C07265=1069.427,-106.395,-57.676,172.308,22.663,154.150
C07266=1069.421,-106.645,-57.666,172.306,22.662,154.150
C07267=1069.415,-106.895,-57.656,172.305,22.661,154.150
C07268=1069.408,-107.144,-57.646,172.303,22.660,154.150
C07269=1069.402,-107.394,-57.636,172.302,22.659,154.150
C07270=1069.396,-107.644,-57.627,172.300,22.658,154.150
C07271=1069.390,-107.894,-57.617,172.299,22.657,154.150
C07272=1069.385,-108.144,-57.607,172.297,22.655,154.150
C07273=1069.378,-108.393,-57.597,172.295,22.654,154.150
C07274=1069.372,-108.643,-57.587,172.294,22.653,154.151
C07275=1069.366,-108.893,-57.578,172.292,22.652,154.151
C07276=1069.360,-109.142,-57.568,172.290,22.651,154.150
C07277=1069.353,-109.392,-57.559,172.289,22.650,154.151
C07278=1069.347,-109.642,-57.549,172.287,22.648,154.151
C07279=1069.341,-109.891,-57.539,172.285,22.648,154.151
C07280=1069.335,-110.141,-57.529,172.284,22.646,154.151
C07281=1069.329,-110.391,-57.519,172.282,22.646,154.151
C07282=1069.323,-110.641,-57.509,172.280,22.644,154.151
C07283=1069.317,-110.891,-57.500,172.279,22.643,154.151
C07284=1069.311,-111.141,-57.490,172.277,22.642,154.151
C07285=1069.304,-111.390,-57.481,172.275,22.641,154.151
C07286=1069.298,-111.640,-57.470,172.273,22.640,154.151
C07287=1069.292,-111.889,-57.461,172.272,22.639,154.151
C07288=1069.286,-112.139,-57.451,172.270,22.638,154.151
C07289=1069.279,-112.389,-57.442,172.268,22.636,154.151
C07290=1069.273,-112.639,-57.432,172.267,22.636,154.151
C07291=1069.267,-112.889,-57.423,172.265,22.634,154.151
C07292=1069.261,-113.138,-57.413,172.263,22.634,154.151
C07293=1069.255,-113.388,-57.403,172.261,22.632,154.151
C07294=1069.250,-113.638,-57.394,172.260,22.631,154.151
C07295=1069.242,-113.918,-57.383,172.258,22.630,154.151
C07296=1069.236,-114.198,-57.373,172.256,22.629,154.151
C07297=1069.229,-114.478,-57.361,172.255,22.628,154.151
C07298=1069.222,-114.758,-57.351,172.253,22.627,154.151
C07299=1069.216,-115.008,-57.341,172.251,22.626,154.152
C07300=1069.210,-115.258,-57.332,172.249,22.625,154.152
C07301=1069.204,-115.508,-57.322,172.248,22.624,154.152
C07302=1069.198,-115.757,-57.312,172.246,22.623,154.152
C07303=1069.191,-116.007,-57.303,172.244,22.622,154.152
C07304=1069.185,-116.257,-57.293,172.243,22.621,154.152
C07305=1069.179,-116.507,-57.284,172.241,22.620,154.152
C07306=1069.173,-116.757,-57.274,172.239,22.619,154.152
C07307=1069.166,-117.006,-57.265,172.237,22.618,154.152
C07308=1069.160,-117.256,-57.256,172.236,22.617,154.152
C07309=1069.154,-117.505,-57.246,172.234,22.616,154.152
C07310=1069.148,-117.755,-57.237,172.232,22.615,154.152
C07311=1069.142,-118.005,-57.227,172.231,22.614,154.152
C07312=1069.136,-118.254,-57.218,172.229,22.613,154.152
C07313=1069.130,-118.504,-57.208,172.227,22.612,154.153
C07314=1069.123,-118.754,-57.199,172.226,22.611,154.152
C07315=1069.117,-119.004,-57.189,172.225,22.610,154.153
C07316=1069.111,-119.254,-57.179,172.223,22.610,154.153
C07317=1069.105,-119.504,-57.171,172.221,22.608,154.153
C07318=1069.100,-119.753,-57.161,172.219,22.607,154.153
C07319=1069.093,-120.003,-57.152,172.218,22.607,154.153
C07320=1069.087,-120.252,-57.143,172.216,22.606,154.153
C07321=1069.080,-120.502,-57.133,172.214,22.605,154.153
C07322=1069.074,-120.752,-57.124,172.212,22.604,154.153
C07323=1069.068,-121.002,-57.114,172.211,22.603,154.153
C07324=1069.062,-121.252,-57.105,172.209,22.602,154.153
C07325=1069.057,-121.501,-57.096,172.207,22.601,154.153
C07326=1069.050,-121.751,-57.087,172.205,22.600,154.153
C07327=1069.043,-122.001,-57.078,172.204,22.599,154.154
C07328=1069.037,-122.250,-57.068,172.202,22.599,154.154
C07329=1069.031,-122.500,-57.058,172.200,22.597,154.154
C07330=1069.025,-122.751,-57.050,172.199,22.597,154.154
C07331=1069.019,-123.000,-57.040,172.197,22.596,154.154
C07332=1069.014,-123.250,-57.031,172.196,22.595,154.154
C07333=1069.007,-123.499,-57.022,172.194,22.594,154.154
C07334=1069.000,-123.749,-57.012,172.192,22.593,154.154
C07335=1068.995,-123.999,-57.003,172.190,22.592,154.154
C07336=1068.988,-124.249,-56.994,172.189,22.592,154.154
C07337=1068.983,-124.498,-56.985,172.187,22.591,154.154
C07338=1068.976,-124.748,-56.976,172.185,22.590,154.155
C07339=1068.970,-124.998,-56.967,172.183,22.589,154.155
C07340=1068.964,-125.248,-56.957,172.182,22.588,154.155
C07341=1068.958,-125.498,-56.948,172.180,22.587,154.155
C07342=1068.951,-125.747,-56.939,172.178,22.586,154.155
C07343=1068.946,-125.997,-56.930,172.177,22.586,154.155
C07344=1068.939,-126.247,-56.921,172.175,22.585,154.155
C07345=1068.933,-126.496,-56.911,172.174,22.584,154.155
C07346=1068.927,-126.747,-56.903,172.172,22.584,154.155
C07347=1068.920,-126.996,-56.893,172.170,22.583,154.155
C07348=1068.915,-127.245,-56.884,172.168,22.582,154.156
C07349=1068.908,-127.495,-56.875,172.166,22.581,154.156
C07350=1068.902,-127.745,-56.866,172.165,22.580,154.156
C07351=1068.897,-127.996,-56.857,172.163,22.580,154.156
C07352=1068.893,-128.247,-56.847,172.161,22.578,154.156
C07353=1068.890,-128.498,-56.836,172.160,22.575,154.155
C07354=1068.890,-128.748,-56.824,172.159,22.573,154.155
C07355=1068.892,-129.001,-56.811,172.158,22.569,154.155
C07356=1068.896,-129.253,-56.798,172.158,22.565,154.154
C07357=1068.901,-129.505,-56.784,172.158,22.560,154.153
C07358=1068.908,-129.755,-56.769,172.158,22.554,154.152
C07359=1068.520,-129.777,-56.938,172.111,22.697,154.184
C07360=1068.512,-129.527,-56.954,172.111,22.703,154.185
C07361=1068.506,-129.276,-56.969,172.111,22.708,154.186
C07362=1068.503,-129.023,-56.982,172.112,22.712,154.187
C07363=1068.501,-128.771,-56.995,172.113,22.716,154.188
C07364=1068.501,-128.520,-57.006,172.114,22.719,154.188
C07365=1068.503,-128.270,-57.017,172.114,22.722,154.188
C07366=1068.507,-128.019,-57.027,172.116,22.723,154.188
C07367=1068.513,-127.768,-57.036,172.117,22.724,154.188
C07368=1068.519,-127.518,-57.046,172.119,22.725,154.188
C07369=1068.525,-127.268,-57.054,172.121,22.726,154.188
C07370=1068.532,-127.018,-57.064,172.123,22.727,154.188
C07371=1068.538,-126.768,-57.073,172.125,22.727,154.188
C07372=1068.543,-126.519,-57.083,172.126,22.728,154.188
C07373=1068.550,-126.269,-57.091,172.128,22.729,154.188
C07374=1068.556,-126.019,-57.100,172.130,22.730,154.188
C07375=1068.562,-125.770,-57.110,172.132,22.730,154.188
C07376=1068.569,-125.519,-57.118,172.133,22.731,154.187
C07377=1068.574,-125.270,-57.127,172.135,22.732,154.187
C07378=1068.581,-125.021,-57.137,172.136,22.732,154.187
C07379=1068.587,-124.771,-57.147,172.138,22.733,154.187
C07380=1068.593,-124.521,-57.155,172.140,22.734,154.187
C07381=1068.600,-124.271,-57.164,172.141,22.735,154.187
C07382=1068.606,-124.021,-57.174,172.143,22.736,154.187
C07383=1068.611,-123.772,-57.183,172.145,22.737,154.187
C07384=1068.617,-123.522,-57.192,172.147,22.738,154.187
C07385=1068.623,-123.272,-57.202,172.149,22.738,154.187
C07386=1068.630,-123.022,-57.211,172.150,22.740,154.187
C07387=1068.636,-122.772,-57.220,172.152,22.740,154.186
C07388=1068.642,-122.523,-57.229,172.154,22.741,154.186
C07389=1068.648,-122.273,-57.238,172.156,22.742,154.186
C07390=1068.654,-122.023,-57.248,172.157,22.743,154.186
C07391=1068.660,-121.773,-57.257,172.159,22.744,154.186
C07392=1068.667,-121.524,-57.266,172.161,22.745,154.186
C07393=1068.673,-121.274,-57.276,172.163,22.746,154.186
C07394=1068.679,-121.024,-57.285,172.164,22.746,154.186
C07395=1068.685,-120.775,-57.294,172.165,22.747,154.186
C07396=1068.691,-120.525,-57.303,172.167,22.748,154.186
C07397=1068.697,-120.275,-57.313,172.169,22.749,154.186
C07398=1068.703,-120.025,-57.323,172.171,22.750,154.186
C07399=1068.709,-119.775,-57.332,172.172,22.751,154.186
C07400=1068.716,-119.526,-57.341,172.174,22.752,154.185
C07401=1068.722,-119.276,-57.351,172.176,22.753,154.185
C07402=1068.728,-119.027,-57.360,172.177,22.754,154.185
C07403=1068.734,-118.777,-57.369,172.179,22.755,154.185
C07404=1068.740,-118.527,-57.378,172.181,22.755,154.185
C07405=1068.746,-118.277,-57.388,172.183,22.757,154.185
C07406=1068.752,-118.027,-57.397,172.184,22.758,154.185
C07407=1068.759,-117.777,-57.407,172.186,22.758,154.185
C07408=1068.765,-117.528,-57.417,172.188,22.760,154.185
C07409=1068.771,-117.278,-57.426,172.190,22.760,154.185
C07410=1068.777,-117.028,-57.436,172.191,22.761,154.185
C07411=1068.783,-116.778,-57.445,172.193,22.763,154.185
C07412=1068.789,-116.528,-57.455,172.194,22.763,154.185
C07413=1068.795,-116.279,-57.464,172.195,22.764,154.185
C07414=1068.801,-116.029,-57.474,172.197,22.765,154.184
C07415=1068.808,-115.780,-57.483,172.199,22.766,154.184
C07416=1068.814,-115.530,-57.492,172.201,22.767,154.184
C07417=1068.820,-115.280,-57.502,172.203,22.768,154.184
C07418=1068.827,-115.031,-57.511,172.204,22.769,154.184
C07419=1068.833,-114.781,-57.521,172.206,22.770,154.184
C07420=1068.840,-114.500,-57.532,172.208,22.771,154.184
C07421=1068.846,-114.220,-57.543,172.210,22.773,154.184
C07422=1068.853,-113.940,-57.554,172.212,22.774,154.184
C07423=1068.860,-113.660,-57.564,172.214,22.775,154.184
C07424=1068.866,-113.410,-57.574,172.215,22.776,154.184
C07425=1068.872,-113.160,-57.584,172.217,22.777,154.184
C07426=1068.878,-112.910,-57.593,172.219,22.778,154.184
C07427=1068.884,-112.661,-57.603,172.220,22.779,154.184
C07428=1068.891,-112.411,-57.612,172.222,22.780,154.184
C07429=1068.897,-112.161,-57.622,172.224,22.781,154.184
C07430=1068.903,-111.911,-57.631,172.226,22.782,154.184
C07431=1068.909,-111.661,-57.641,172.227,22.783,154.184
C07432=1068.916,-111.412,-57.651,172.229,22.784,154.184
C07433=1068.922,-111.162,-57.661,172.231,22.786,154.184
C07434=1068.927,-110.912,-57.671,172.232,22.787,154.183
C07435=1068.933,-110.662,-57.681,172.234,22.788,154.183
C07436=1068.939,-110.413,-57.690,172.235,22.788,154.183
C07437=1068.946,-110.163,-57.700,172.236,22.790,154.183
C07438=1068.952,-109.913,-57.709,172.238,22.790,154.183
C07439=1068.958,-109.664,-57.720,172.240,22.792,154.183
C07440=1068.964,-109.414,-57.729,172.242,22.793,154.183
C07441=1068.971,-109.164,-57.739,172.243,22.794,154.183
C07442=1068.977,-108.915,-57.748,172.245,22.795,154.183
C07443=1068.983,-108.665,-57.758,172.247,22.796,154.183
C07444=1068.988,-108.415,-57.768,172.248,22.797,154.183
C07445=1068.995,-108.165,-57.778,172.250,22.799,154.183
C07446=1069.001,-107.916,-57.788,172.252,22.799,154.183
C07447=1069.007,-107.666,-57.797,172.253,22.801,154.183
C07448=1069.013,-107.416,-57.807,172.255,22.802,154.183
C07449=1069.020,-107.167,-57.817,172.257,22.803,154.183
C07450=1069.025,-106.917,-57.827,172.258,22.804,154.183
C07451=1069.031,-106.667,-57.837,172.260,22.805,154.183
C07452=1069.038,-106.417,-57.847,172.262,22.806,154.183
C07453=1069.044,-106.168,-57.857,172.263,22.808,154.183
C07454=1069.050,-105.918,-57.866,172.265,22.809,154.183
C07455=1069.056,-105.668,-57.877,172.267,22.810,154.183
C07456=1069.062,-105.418,-57.886,172.268,22.811,154.183
C07457=1069.068,-105.169,-57.896,172.270,22.812,154.183
C07458=1069.075,-104.919,-57.906,172.272,22.814,154.183
C07459=1069.080,-104.669,-57.916,172.273,22.815,154.183
C07460=1069.086,-104.420,-57.926,172.275,22.816,154.183
C07461=1069.093,-104.170,-57.936,172.277,22.817,154.183
C07462=1069.098,-103.920,-57.946,172.278,22.818,154.183
C07463=1069.105,-103.671,-57.956,172.280,22.820,154.183
C07464=1069.111,-103.420,-57.966,172.282,22.821,154.183
C07465=1069.117,-103.171,-57.976,172.283,22.822,154.183
C07466=1069.123,-102.921,-57.987,172.285,22.823,154.183
C07467=1069.129,-102.671,-57.996,172.287,22.825,154.183
C07468=1069.136,-102.422,-58.006,172.288,22.826,154.183
C07469=1069.141,-102.172,-58.017,172.290,22.827,154.183
C07470=1069.147,-101.922,-58.026,172.292,22.829,154.183
C07471=1069.154,-101.672,-58.036,172.293,22.829,154.183
C07472=1069.159,-101.423,-58.047,172.295,22.831,154.183
C07473=1069.166,-101.173,-58.056,172.297,22.832,154.183
C07474=1069.172,-100.924,-58.067,172.298,22.833,154.183
C07475=1069.177,-100.674,-58.077,172.300,22.835,154.183
C07476=1069.184,-100.423,-58.087,172.301,22.836,154.183
C07477=1069.191,-100.174,-58.097,172.303,22.837,154.183
C07478=1069.197,-99.924,-58.107,172.305,22.839,154.183
C07479=1069.203,-99.675,-58.117,172.306,22.839,154.183
C07480=1069.209,-99.425,-58.127,172.308,22.841,154.183
C07481=1069.215,-99.176,-58.138,172.310,22.842,154.183
C07482=1069.221,-98.926,-58.147,172.311,22.843,154.183
C07483=1069.228,-98.676,-58.158,172.313,22.845,154.183
C07484=1069.234,-98.394,-58.169,172.315,22.846,154.183
C07485=1069.241,-98.111,-58.181,172.316,22.847,154.183
C07486=1069.248,-97.828,-58.192,172.318,22.849,154.183
C07487=1069.255,-97.546,-58.204,172.320,22.851,154.183
C07488=1069.262,-97.296,-58.214,172.322,22.852,154.183
C07489=1069.267,-97.046,-58.225,172.324,22.853,154.183
C07490=1069.274,-96.797,-58.235,172.325,22.855,154.183
C07491=1069.279,-96.547,-58.245,172.327,22.856,154.183
C07492=1069.286,-96.298,-58.255,172.328,22.858,154.183
C07493=1069.291,-96.048,-58.265,172.330,22.859,154.183
C07494=1069.297,-95.798,-58.276,172.331,22.860,154.183
C07495=1069.303,-95.548,-58.286,172.333,22.862,154.183
C07496=1069.309,-95.299,-58.297,172.335,22.863,154.183
C07497=1069.315,-95.048,-58.307,172.336,22.864,154.183
C07498=1069.321,-94.799,-58.318,172.338,22.866,154.183
C07499=1069.328,-94.550,-58.328,172.340,22.867,154.183
C07500=1069.333,-94.300,-58.338,172.341,22.868,154.183
C07501=1069.340,-94.050,-58.348,172.343,22.870,154.183
C07502=1069.345,-93.800,-58.358,172.344,22.872,154.183
C07503=1069.351,-93.551,-58.369,172.346,22.873,154.183
C07504=1069.358,-93.301,-58.380,172.347,22.874,154.183
C07505=1069.363,-93.051,-58.390,172.349,22.876,154.183
C07506=1069.370,-92.802,-58.400,172.351,22.877,154.183
C07507=1069.375,-92.552,-58.411,172.352,22.878,154.183
C07508=1069.382,-92.302,-58.421,172.354,22.880,154.183
C07509=1069.388,-92.052,-58.432,172.355,22.882,154.183
C07510=1069.394,-91.803,-58.443,172.357,22.883,154.183
C07511=1069.400,-91.553,-58.453,172.359,22.884,154.183
C07512=1069.406,-91.303,-58.463,172.360,22.886,154.183
C07513=1069.412,-91.054,-58.474,172.362,22.887,154.183
C07514=1069.418,-90.803,-58.484,172.363,22.889,154.184
C07515=1069.424,-90.554,-58.495,172.365,22.890,154.184
C07516=1069.430,-90.305,-58.505,172.367,22.891,154.184
C07517=1069.436,-90.055,-58.516,172.368,22.893,154.184
C07518=1069.442,-89.805,-58.526,172.370,22.894,154.184
C07519=1069.449,-89.555,-58.537,172.371,22.896,154.184
C07520=1069.454,-89.306,-58.548,172.373,22.897,154.184
C07521=1069.461,-89.056,-58.558,172.374,22.899,154.184
C07522=1069.466,-88.806,-58.568,172.376,22.900,154.184
C07523=1069.473,-88.556,-58.580,172.378,22.902,154.184
C07524=1069.479,-88.307,-58.590,172.379,22.903,154.184
C07525=1069.485,-88.057,-58.600,172.381,22.905,154.184
C07526=1069.491,-87.808,-58.610,172.382,22.906,154.184
C07527=1069.497,-87.558,-58.622,172.384,22.908,154.184
C07528=1069.503,-87.308,-58.633,172.385,22.909,154.184
C07529=1069.510,-87.059,-58.643,172.387,22.910,154.184
C07530=1069.516,-86.808,-58.653,172.389,22.912,154.184
C07531=1069.521,-86.559,-58.664,172.390,22.914,154.184
C07532=1069.528,-86.309,-58.675,172.392,22.915,154.184
C07533=1069.534,-86.060,-58.685,172.393,22.916,154.184
C07534=1069.540,-85.810,-58.697,172.395,22.918,154.184
C07535=1069.546,-85.561,-58.707,172.396,22.920,154.185
C07536=1069.552,-85.310,-58.717,172.398,22.921,154.185
C07537=1069.558,-85.060,-58.728,172.400,22.922,154.185
C07538=1069.565,-84.811,-58.739,172.401,22.924,154.185
C07539=1069.570,-84.562,-58.749,172.403,22.925,154.185
C07540=1069.577,-84.311,-58.761,172.404,22.927,154.185
C07541=1069.583,-84.062,-58.771,172.406,22.929,154.185
C07542=1069.589,-83.813,-58.782,172.407,22.930,154.185
C07543=1069.595,-83.563,-58.793,172.409,22.931,154.185
C07544=1069.602,-83.313,-58.803,172.411,22.934,154.185
C07545=1069.607,-83.063,-58.814,172.413,22.935,154.185
C07546=1069.614,-82.813,-58.825,172.415,22.936,154.185
C07547=1069.620,-82.564,-58.835,172.416,22.938,154.185
C07548=1069.627,-82.284,-58.847,172.418,22.940,154.185
C07549=1069.633,-82.003,-58.860,172.419,22.941,154.185
C07550=1069.640,-81.723,-58.872,172.421,22.943,154.185
C07551=1069.647,-81.443,-58.884,172.423,22.945,154.186
C07552=1069.654,-81.193,-58.895,172.425,22.946,154.186
C07553=1069.660,-80.944,-58.906,172.426,22.948,154.186
C07554=1069.666,-80.694,-58.916,172.428,22.950,154.186
C07555=1069.673,-80.444,-58.927,172.429,22.951,154.186
C07556=1069.678,-80.195,-58.938,172.431,22.953,154.186
C07557=1069.685,-79.945,-58.949,172.433,22.954,154.186
C07558=1069.691,-79.695,-58.960,172.434,22.956,154.186
C07559=1069.696,-79.446,-58.971,172.436,22.957,154.186
C07560=1069.703,-79.195,-58.982,172.437,22.959,154.186
C07561=1069.709,-78.946,-58.993,172.439,22.961,154.186
C07562=1069.715,-78.697,-59.003,172.440,22.962,154.186
C07563=1069.721,-78.446,-59.015,172.442,22.964,154.186
C07564=1069.727,-78.197,-59.025,172.443,22.966,154.187
C07565=1069.733,-77.948,-59.036,172.445,22.967,154.187
C07566=1069.739,-77.697,-59.048,172.446,22.969,154.187
C07567=1069.745,-77.448,-59.059,172.448,22.970,154.187
C07568=1069.751,-77.198,-59.070,172.449,22.972,154.187
C07569=1069.757,-76.949,-59.081,172.451,22.974,154.187
C07570=1069.763,-76.699,-59.092,172.452,22.975,154.187
C07571=1069.769,-76.449,-59.103,172.454,22.977,154.187
C07572=1069.776,-76.200,-59.114,172.455,22.979,154.187
C07573=1069.782,-75.950,-59.125,172.458,22.981,154.187
C07574=1069.788,-75.700,-59.136,172.459,22.982,154.187
C07575=1069.794,-75.451,-59.147,172.461,22.984,154.187
C07576=1069.800,-75.201,-59.159,172.462,22.986,154.188
C07577=1069.806,-74.952,-59.170,172.464,22.987,154.188
C07578=1069.812,-74.701,-59.181,172.465,22.989,154.188
C07579=1069.818,-74.452,-59.192,172.467,22.991,154.188
C07580=1069.824,-74.202,-59.203,172.468,22.992,154.188
C07581=1069.830,-73.952,-59.214,172.470,22.994,154.188
C07582=1069.836,-73.703,-59.225,172.472,22.996,154.188
C07583=1069.842,-73.453,-59.237,172.473,22.998,154.188
C07584=1069.848,-73.204,-59.248,172.474,22.999,154.188
C07585=1069.855,-72.954,-59.259,172.476,23.001,154.189
C07586=1069.860,-72.704,-59.270,172.478,23.003,154.189
C07587=1069.866,-72.455,-59.282,172.479,23.005,154.189
C07588=1069.872,-72.205,-59.293,172.480,23.006,154.189
C07589=1069.878,-71.955,-59.304,172.482,23.008,154.189
C07590=1069.884,-71.705,-59.315,172.483,23.010,154.189
C07591=1069.890,-71.456,-59.327,172.485,23.012,154.189
C07592=1069.895,-71.206,-59.338,172.486,23.013,154.189
C07593=1069.901,-70.956,-59.350,172.488,23.015,154.189
C07594=1069.907,-70.707,-59.361,172.489,23.017,154.190
C07595=1069.914,-70.457,-59.372,172.491,23.019,154.190
C07596=1069.919,-70.208,-59.383,172.493,23.021,154.190
C07597=1069.926,-69.957,-59.394,172.495,23.023,154.190
C07598=1069.931,-69.708,-59.407,172.496,23.025,154.190
C07599=1069.937,-69.459,-59.418,172.498,23.026,154.190
C07600=1069.943,-69.209,-59.429,172.499,23.028,154.190
C07601=1069.949,-68.960,-59.440,172.501,23.030,154.190
C07602=1069.956,-68.709,-59.452,172.502,23.032,154.190
C07603=1069.961,-68.460,-59.463,172.504,23.033,154.191
C07604=1069.967,-68.210,-59.475,172.505,23.035,154.191
C07605=1069.973,-67.961,-59.486,172.507,23.037,154.191
C07606=1069.979,-67.710,-59.497,172.508,23.039,154.191
C07607=1069.985,-67.462,-59.509,172.510,23.040,154.191
C07608=1069.991,-67.211,-59.521,172.511,23.042,154.191
C07609=1069.997,-66.962,-59.532,172.512,23.044,154.191
C07610=1070.003,-66.712,-59.543,172.514,23.046,154.192
C07611=1070.009,-66.463,-59.554,172.515,23.048,154.192
C07612=1070.016,-66.184,-59.568,172.518,23.050,154.192
C07613=1070.022,-65.907,-59.580,172.519,23.052,154.192
C07614=1070.029,-65.629,-59.594,172.521,23.054,154.192
C07615=1070.036,-65.350,-59.606,172.522,23.056,154.192
C07616=1070.042,-65.101,-59.617,172.524,23.058,154.192
C07617=1070.048,-64.851,-59.629,172.526,23.060,154.192
C07618=1070.054,-64.602,-59.641,172.527,23.062,154.193
C07619=1070.060,-64.351,-59.652,172.529,23.064,154.193
C07620=1070.066,-64.103,-59.664,172.530,23.066,154.193
C07621=1070.073,-63.852,-59.675,172.532,23.068,154.193
C07622=1070.078,-63.603,-59.687,172.533,23.069,154.193
C07623=1070.084,-63.353,-59.698,172.535,23.071,154.193
C07624=1070.091,-63.103,-59.710,172.536,23.073,154.193
C07625=1070.097,-62.854,-59.721,172.538,23.075,154.193
C07626=1070.102,-62.604,-59.734,172.539,23.076,154.194
C07627=1070.108,-62.355,-59.745,172.541,23.078,154.194
C07628=1070.115,-62.105,-59.757,172.542,23.080,154.194
C07629=1070.120,-61.855,-59.768,172.543,23.082,154.194
C07630=1070.127,-61.606,-59.780,172.545,23.084,154.194
C07631=1070.133,-61.355,-59.791,172.546,23.086,154.194
C07632=1070.139,-61.107,-59.803,172.548,23.088,154.195
C07633=1070.144,-60.856,-59.815,172.550,23.090,154.195
C07634=1070.151,-60.607,-59.826,172.552,23.092,154.195
C07635=1070.157,-60.358,-59.838,172.553,23.094,154.195
C07636=1070.164,-60.107,-59.849,172.555,23.096,154.195
C07637=1070.169,-59.858,-59.862,172.556,23.098,154.195
C07638=1070.175,-59.608,-59.873,172.557,23.099,154.195
C07639=1070.182,-59.358,-59.885,172.559,23.101,154.195
C07640=1070.187,-59.109,-59.897,172.560,23.103,154.196
C07641=1070.193,-58.859,-59.908,172.562,23.105,154.196
C07642=1070.200,-58.610,-59.920,172.563,23.107,154.196
C07643=1070.205,-58.360,-59.932,172.565,23.109,154.196
C07644=1070.212,-58.110,-59.944,172.566,23.111,154.196
C07645=1070.218,-57.861,-59.955,172.568,23.113,154.196
C07646=1070.224,-57.611,-59.967,172.569,23.115,154.197
C07647=1070.230,-57.361,-59.979,172.571,23.116,154.197
C07648=1070.236,-57.112,-59.991,172.572,23.118,154.197
C07649=1070.243,-56.863,-60.003,172.574,23.121,154.197
C07650=1070.248,-56.612,-60.014,172.576,23.122,154.197
C07651=1070.254,-56.363,-60.026,172.577,23.124,154.197
C07652=1070.261,-56.114,-60.038,172.579,23.126,154.197
C07653=1070.267,-55.863,-60.050,172.580,23.128,154.198
C07654=1070.273,-55.614,-60.062,172.582,23.130,154.198
C07655=1070.279,-55.365,-60.073,172.583,23.132,154.198
C07656=1070.285,-55.114,-60.085,172.585,23.134,154.198
C07657=1070.292,-54.865,-60.097,172.586,23.136,154.198
C07658=1070.298,-54.616,-60.109,172.587,23.138,154.198
C07659=1070.304,-54.366,-60.121,172.589,23.139,154.198
C07660=1070.310,-54.116,-60.133,172.590,23.141,154.199
C07661=1070.316,-53.866,-60.145,172.592,23.143,154.199
C07662=1070.322,-53.617,-60.157,172.593,23.145,154.199
C07663=1070.328,-53.368,-60.169,172.595,23.147,154.199
C07664=1070.334,-53.118,-60.181,172.597,23.149,154.199
C07665=1070.341,-52.867,-60.193,172.599,23.151,154.199
C07666=1070.347,-52.619,-60.204,172.600,23.154,154.200
C07667=1070.353,-52.369,-60.217,172.601,23.155,154.200
C07668=1070.359,-52.119,-60.229,172.603,23.157,154.200
C07669=1070.366,-51.870,-60.241,172.604,23.159,154.200
C07670=1070.371,-51.620,-60.253,172.606,23.161,154.200
C07671=1070.378,-51.370,-60.264,172.607,23.163,154.200
C07672=1070.384,-51.120,-60.277,172.609,23.165,154.200
C07673=1070.390,-50.871,-60.289,172.610,23.167,154.201
C07674=1070.397,-50.621,-60.300,172.611,23.169,154.201
C07675=1070.402,-50.372,-60.313,172.613,23.170,154.201
C07676=1070.409,-50.095,-60.326,172.615,23.173,154.201
C07677=1070.415,-49.818,-60.340,172.617,23.175,154.201
C07678=1070.423,-49.542,-60.353,172.618,23.178,154.201
C07679=1070.429,-49.265,-60.367,172.620,23.180,154.202
C07680=1070.435,-49.015,-60.379,172.621,23.182,154.202
C07681=1070.441,-48.766,-60.391,172.623,23.184,154.202
C07682=1070.447,-48.516,-60.403,172.624,23.186,154.202
C07683=1070.453,-48.266,-60.416,172.626,23.188,154.202
C07684=1070.459,-48.017,-60.428,172.627,23.190,154.203
C07685=1070.465,-47.767,-60.440,172.629,23.192,154.203
C07686=1070.470,-47.517,-60.453,172.630,23.195,154.203
C07687=1070.477,-47.268,-60.465,172.631,23.197,154.203
C07688=1070.483,-47.018,-60.477,172.633,23.198,154.203
C07689=1070.488,-46.769,-60.489,172.634,23.200,154.203
C07690=1070.495,-46.519,-60.501,172.636,23.203,154.204
C07691=1070.501,-46.269,-60.514,172.637,23.205,154.204
C07692=1070.507,-46.019,-60.526,172.638,23.206,154.204
C07693=1070.513,-45.771,-60.538,172.641,23.209,154.204
C07694=1070.519,-45.521,-60.551,172.642,23.211,154.204
C07695=1070.525,-45.271,-60.563,172.644,23.213,154.205
C07696=1070.531,-45.021,-60.575,172.645,23.216,154.205
C07697=1070.537,-44.771,-60.588,172.646,23.217,154.205
C07698=1070.543,-44.522,-60.600,172.648,23.219,154.205
C07699=1070.548,-44.272,-60.612,172.649,23.222,154.205
C07700=1070.555,-44.023,-60.624,172.651,23.224,154.206
C07701=1070.561,-43.773,-60.637,172.652,23.225,154.206
C07702=1070.567,-43.523,-60.649,172.653,23.228,154.206
C07703=1070.574,-43.273,-60.661,172.655,23.230,154.206
C07704=1070.579,-43.024,-60.674,172.656,23.232,154.206
C07705=1070.585,-42.774,-60.686,172.657,23.234,154.207
C07706=1070.591,-42.524,-60.699,172.660,23.236,154.207
C07707=1070.598,-42.276,-60.711,172.661,23.239,154.207
C07708=1070.604,-42.026,-60.724,172.663,23.241,154.207
C07709=1070.609,-41.776,-60.736,172.664,23.243,154.207
C07710=1070.616,-41.527,-60.748,172.665,23.245,154.208
C07711=1070.621,-41.277,-60.761,172.667,23.247,154.208
C07712=1070.627,-41.027,-60.773,172.668,23.249,154.208
C07713=1070.633,-40.777,-60.786,172.670,23.251,154.208
C07714=1070.640,-40.528,-60.798,172.671,23.253,154.208
C07715=1070.646,-40.278,-60.811,172.672,23.255,154.209
C07716=1070.652,-40.028,-60.824,172.674,23.257,154.209
C07717=1070.658,-39.779,-60.836,172.675,23.259,154.209
C07718=1070.664,-39.530,-60.848,172.677,23.262,154.209
C07719=1070.670,-39.280,-60.861,172.679,23.264,154.209
C07720=1070.676,-39.031,-60.873,172.680,23.266,154.209
C07721=1070.682,-38.781,-60.886,172.682,23.268,154.210
C07722=1070.688,-38.531,-60.899,172.683,23.271,154.210
C07723=1070.694,-38.281,-60.911,172.684,23.273,154.210
C07724=1070.701,-38.032,-60.924,172.686,23.275,154.210
C07725=1070.707,-37.782,-60.936,172.687,23.277,154.210
C07726=1070.713,-37.532,-60.949,172.688,23.279,154.211
C07727=1070.718,-37.283,-60.961,172.690,23.281,154.211
C07728=1070.724,-37.034,-60.974,172.691,23.284,154.211
C07729=1070.730,-36.784,-60.987,172.693,23.285,154.211
C07730=1070.736,-36.534,-60.999,172.694,23.288,154.212
C07731=1070.742,-36.285,-61.013,172.696,23.290,154.212
C07732=1070.748,-36.035,-61.025,172.698,23.293,154.212
C07733=1070.754,-35.785,-61.038,172.699,23.294,154.212
C07734=1070.760,-35.536,-61.051,172.700,23.297,154.212
C07735=1070.766,-35.286,-61.064,172.702,23.299,154.213
C07736=1070.771,-35.037,-61.076,172.703,23.301,154.213
C07737=1070.778,-34.787,-61.089,172.704,23.304,154.213
C07738=1070.783,-34.538,-61.102,172.706,23.305,154.213
C07739=1070.789,-34.288,-61.114,172.707,23.308,154.214
C07740=1070.796,-34.011,-61.129,172.708,23.310,154.214
C07741=1070.803,-33.735,-61.143,172.711,23.313,154.214
C07742=1070.810,-33.459,-61.157,172.712,23.315,154.214
C07743=1070.816,-33.182,-61.171,172.713,23.317,154.214
C07744=1070.823,-32.933,-61.184,172.715,23.320,154.215
C07745=1070.828,-32.683,-61.197,172.717,23.322,154.215
C07746=1070.835,-32.433,-61.210,172.718,23.325,154.215
C07747=1070.841,-32.184,-61.223,172.720,23.326,154.215
C07748=1070.846,-31.934,-61.235,172.721,23.329,154.216
C07749=1070.852,-31.685,-61.248,172.722,23.331,154.216
C07750=1070.858,-31.435,-61.261,172.724,23.333,154.216
C07751=1070.864,-31.186,-61.274,172.725,23.336,154.216
C07752=1070.870,-30.936,-61.286,172.727,23.337,154.216
C07753=1070.876,-30.687,-61.300,172.728,23.340,154.217
C07754=1070.882,-30.437,-61.312,172.729,23.342,154.217
C07755=1070.888,-30.188,-61.326,172.731,23.344,154.217
C07756=1070.894,-29.938,-61.338,172.732,23.347,154.217
C07757=1070.901,-29.688,-61.351,172.734,23.349,154.218
C07758=1070.906,-29.439,-61.364,172.736,23.351,154.218
C07759=1070.913,-29.189,-61.377,172.737,23.353,154.218
C07760=1070.919,-28.939,-61.390,172.738,23.356,154.218
C07761=1070.925,-28.689,-61.403,172.740,23.358,154.218
C07762=1070.931,-28.440,-61.416,172.741,23.360,154.219
C07763=1070.938,-28.190,-61.429,172.742,23.362,154.219
C07764=1070.943,-27.940,-61.442,172.744,23.365,154.219
C07765=1070.949,-27.691,-61.456,172.745,23.367,154.219
C07766=1070.955,-27.441,-61.468,172.747,23.369,154.220
C07767=1070.961,-27.192,-61.481,172.748,23.371,154.220
C07768=1070.967,-26.942,-61.495,172.749,23.373,154.220
C07769=1070.973,-26.693,-61.507,172.752,23.376,154.220
C07770=1070.979,-26.443,-61.521,172.753,23.378,154.220
C07771=1070.985,-26.193,-61.533,172.754,23.380,154.221
C07772=1070.991,-25.944,-61.547,172.756,23.383,154.221
C07773=1070.997,-25.695,-61.560,172.757,23.385,154.221
C07774=1071.003,-25.445,-61.573,172.758,23.387,154.221
C07775=1071.009,-25.195,-61.586,172.760,23.390,154.222
C07776=1071.014,-24.945,-61.599,172.761,23.392,154.222
C07777=1071.020,-24.696,-61.612,172.762,23.394,154.222
C07778=1071.027,-24.447,-61.626,172.764,23.396,154.222
C07779=1071.033,-24.197,-61.638,172.765,23.399,154.223
C07780=1071.038,-23.947,-61.652,172.766,23.401,154.223
C07781=1071.044,-23.698,-61.665,172.769,23.404,154.223
C07782=1071.050,-23.448,-61.678,172.770,23.406,154.223
C07783=1071.056,-23.199,-61.691,172.771,23.408,154.224
C07784=1071.062,-22.949,-61.705,172.773,23.411,154.224
C07785=1071.069,-22.699,-61.719,172.774,23.413,154.224
C07786=1071.075,-22.449,-61.731,172.775,23.415,154.224
C07787=1071.081,-22.200,-61.745,172.777,23.417,154.225
C07788=1071.086,-21.951,-61.758,172.778,23.420,154.225
C07789=1071.093,-21.701,-61.772,172.779,23.422,154.225
C07790=1071.098,-21.451,-61.784,172.781,23.425,154.225
C07791=1071.104,-21.202,-61.798,172.782,23.426,154.226
C07792=1071.110,-20.953,-61.811,172.784,23.429,154.226
C07793=1071.116,-20.703,-61.825,172.786,23.432,154.226
C07794=1071.122,-20.453,-61.838,172.787,23.434,154.226
C07795=1071.128,-20.204,-61.851,172.788,23.437,154.227
C07796=1071.135,-19.954,-61.865,172.790,23.438,154.227
C07797=1071.141,-19.705,-61.878,172.791,23.441,154.227
C07798=1071.146,-19.455,-61.892,172.792,23.443,154.227
C07799=1071.152,-19.205,-61.904,172.794,23.446,154.228
C07800=1071.158,-18.956,-61.918,172.795,23.448,154.228
C07801=1071.164,-18.706,-61.932,172.796,23.450,154.228
C07802=1071.170,-18.457,-61.945,172.798,23.452,154.228
C07803=1071.177,-18.207,-61.958,172.799,23.455,154.229
C07804=1071.182,-17.930,-61.973,172.801,23.458,154.229
C07805=1071.190,-17.653,-61.988,172.802,23.460,154.229
C07806=1071.196,-17.375,-62.003,172.804,23.462,154.229
C07807=1071.203,-17.098,-62.018,172.806,23.465,154.230
C07808=1071.210,-16.849,-62.031,172.807,23.468,154.230
C07809=1071.215,-16.599,-62.045,172.809,23.470,154.230
C07810=1071.221,-16.350,-62.058,172.810,23.472,154.231
C07811=1071.227,-16.101,-62.072,172.811,23.475,154.231
C07812=1071.233,-15.850,-62.085,172.813,23.477,154.231
C07813=1071.239,-15.601,-62.099,172.814,23.479,154.231
C07814=1071.245,-15.351,-62.112,172.815,23.482,154.231
C07815=1071.251,-15.102,-62.126,172.817,23.484,154.232
C07816=1071.257,-14.853,-62.139,172.819,23.487,154.232
C07817=1071.263,-14.603,-62.153,172.820,23.489,154.232
C07818=1071.270,-14.353,-62.166,172.821,23.492,154.233
C07819=1071.275,-14.104,-62.180,172.823,23.494,154.233
C07820=1071.281,-13.854,-62.194,172.824,23.496,154.233
C07821=1071.287,-13.605,-62.207,172.825,23.498,154.233
C07822=1071.292,-13.355,-62.221,172.827,23.501,154.234
C07823=1071.299,-13.105,-62.235,172.828,23.503,154.234
C07824=1071.305,-12.856,-62.249,172.829,23.506,154.234
C07825=1071.311,-12.606,-62.262,172.831,23.508,154.234
C07826=1071.316,-12.357,-62.276,172.832,23.510,154.235
C07827=1071.323,-12.107,-62.289,172.833,23.513,154.235
C07828=1071.328,-11.858,-62.303,172.836,23.516,154.235
C07829=1071.334,-11.608,-62.317,172.837,23.518,154.235
C07830=1071.340,-11.358,-62.331,172.838,23.520,154.236
C07831=1071.346,-11.109,-62.344,172.839,23.523,154.236
C07832=1071.352,-10.859,-62.358,172.841,23.525,154.236
C07833=1071.358,-10.609,-62.372,172.842,23.528,154.237
C07834=1071.365,-10.361,-62.386,172.843,23.530,154.237
C07835=1071.370,-10.111,-62.400,172.845,23.532,154.237
C07836=1071.376,-9.861,-62.414,172.846,23.534,154.237
C07837=1071.382,-9.611,-62.427,172.847,23.537,154.238
C07838=1071.388,-9.362,-62.441,172.849,23.539,154.238
C07839=1071.394,-9.113,-62.454,172.851,23.542,154.238
C07840=1071.399,-8.863,-62.468,172.852,23.544,154.238
C07841=1071.406,-8.613,-62.482,172.854,23.547,154.239
C07842=1071.412,-8.364,-62.497,172.855,23.549,154.239
C07843=1071.418,-8.115,-62.510,172.856,23.552,154.239
C07844=1071.424,-7.865,-62.524,172.858,23.554,154.239
C07845=1071.430,-7.615,-62.538,172.859,23.557,154.240
C07846=1071.436,-7.366,-62.551,172.860,23.559,154.240
C07847=1071.442,-7.116,-62.565,172.861,23.561,154.240
C07848=1071.448,-6.867,-62.580,172.863,23.564,154.241
C07849=1071.454,-6.617,-62.593,172.864,23.566,154.241
C07850=1071.460,-6.368,-62.607,172.866,23.569,154.241
C07851=1071.465,-6.118,-62.621,172.868,23.571,154.241
C07852=1071.472,-5.868,-62.635,172.869,23.574,154.242
C07853=1071.478,-5.619,-62.649,172.870,23.576,154.242
C07854=1071.484,-5.370,-62.662,172.872,23.579,154.242
C07855=1071.490,-5.120,-62.677,172.873,23.581,154.243
C07856=1071.495,-4.870,-62.691,172.874,23.583,154.243
C07857=1071.502,-4.621,-62.705,172.875,23.586,154.243
C07858=1071.508,-4.371,-62.719,172.877,23.588,154.243
C07859=1071.514,-4.122,-62.733,172.878,23.590,154.244
C07860=1071.520,-3.872,-62.746,172.880,23.593,154.244
C07861=1071.526,-3.623,-62.761,172.881,23.595,154.244
C07862=1071.532,-3.373,-62.775,172.883,23.598,154.244
C07863=1071.538,-3.123,-62.788,172.884,23.600,154.245
C07864=1071.544,-2.874,-62.803,172.886,23.603,154.245
C07865=1071.550,-2.625,-62.817,172.887,23.606,154.245
C07866=1071.555,-2.375,-62.831,172.888,23.608,154.246
C07867=1071.562,-2.125,-62.846,172.890,23.610,154.246
C07868=1071.568,-1.846,-62.861,172.891,23.613,154.246
C07869=1071.574,-1.568,-62.876,172.893,23.616,154.246
C07870=1071.581,-1.289,-62.893,172.894,23.618,154.247
C07871=1071.587,-1.010,-62.908,172.895,23.621,154.247
C07872=1071.594,-0.761,-62.923,172.897,23.624,154.247
C07873=1071.599,-0.511,-62.937,172.899,23.627,154.248
C07874=1071.605,-0.262,-62.951,172.900,23.629,154.248
C07875=1071.611,-0.012,-62.966,172.902,23.631,154.248
C07876=1071.617,0.238,-62.979,172.903,23.634,154.249
C07877=1071.622,0.487,-62.994,172.904,23.637,154.249
C07878=1071.629,0.737,-63.008,172.905,23.639,154.249
C07879=1071.634,0.986,-63.023,172.907,23.642,154.249
C07880=1071.640,1.235,-63.037,172.908,23.644,154.250
C07881=1071.647,1.485,-63.050,172.909,23.646,154.250
C07882=1071.652,1.734,-63.065,172.911,23.649,154.250
C07883=1071.658,1.984,-63.079,172.912,23.651,154.251
C07884=1071.664,2.234,-63.094,172.914,23.654,154.251
C07885=1071.670,2.483,-63.108,172.915,23.657,154.251
C07886=1071.676,2.733,-63.123,172.917,23.659,154.252
C07887=1071.682,2.982,-63.136,172.918,23.662,154.252
C07888=1071.687,3.231,-63.151,172.919,23.664,154.252
C07889=1071.693,3.482,-63.165,172.921,23.667,154.252
C07890=1071.699,3.731,-63.180,172.922,23.669,154.253
C07891=1071.705,3.980,-63.194,172.923,23.671,154.253
C07892=1071.711,4.230,-63.209,172.925,23.674,154.253
C07893=1071.717,4.479,-63.222,172.926,23.677,154.254
C07894=1071.723,4.729,-63.237,172.927,23.679,154.254
C07895=1071.729,4.978,-63.252,172.929,23.682,154.254
C07896=1071.735,5.228,-63.266,172.931,23.684,154.254
C07897=1071.741,5.477,-63.281,172.932,23.687,154.255
C07898=1071.746,5.727,-63.295,172.933,23.689,154.255
C07899=1071.752,5.976,-63.310,172.934,23.692,154.255
C07900=1071.758,6.226,-63.324,172.936,23.694,154.256
C07901=1071.764,6.476,-63.338,172.937,23.697,154.256
C07902=1071.770,6.725,-63.353,172.938,23.699,154.256
C07903=1071.776,6.975,-63.367,172.940,23.702,154.257
C07904=1071.782,7.224,-63.382,172.941,23.704,154.257
C07905=1071.788,7.474,-63.397,172.942,23.707,154.257
C07906=1071.794,7.723,-63.411,172.944,23.709,154.257
C07907=1071.800,7.973,-63.426,172.946,23.712,154.258
C07908=1071.806,8.222,-63.440,172.947,23.715,154.258
C07909=1071.812,8.472,-63.454,172.948,23.717,154.258
C07910=1071.818,8.721,-63.469,172.950,23.720,154.259
C07911=1071.824,8.971,-63.484,172.951,23.722,154.259
C07912=1071.830,9.220,-63.498,172.952,23.724,154.259
C07913=1071.836,9.470,-63.513,172.954,23.727,154.259
C07914=1071.842,9.719,-63.527,172.955,23.729,154.260
C07915=1071.848,9.969,-63.542,172.956,23.732,154.260
C07916=1071.854,10.218,-63.556,172.958,23.735,154.260
C07917=1071.860,10.468,-63.571,172.960,23.737,154.261
C07918=1071.866,10.717,-63.586,172.961,23.740,154.261
C07919=1071.872,10.967,-63.600,172.962,23.742,154.261
C07920=1071.878,11.216,-63.614,172.964,23.745,154.261
C07921=1071.884,11.466,-63.629,172.965,23.747,154.262
C07922=1071.890,11.714,-63.644,172.966,23.749,154.262
C07923=1071.896,11.965,-63.658,172.968,23.752,154.262
C07924=1071.902,12.214,-63.673,172.969,23.755,154.263
C07925=1071.908,12.463,-63.688,172.970,23.757,154.263
C07926=1071.915,12.713,-63.703,172.971,23.759,154.263
C07927=1071.920,12.963,-63.717,172.974,23.762,154.264
C07928=1071.926,13.212,-63.732,172.975,23.765,154.264
C07929=1071.932,13.461,-63.746,172.976,23.767,154.264
C07930=1071.939,13.711,-63.761,172.978,23.769,154.264
C07931=1071.945,13.961,-63.776,172.979,23.772,154.265
C07932=1071.951,14.241,-63.793,172.980,23.775,154.265
C07933=1071.958,14.522,-63.809,172.982,23.778,154.265
C07934=1071.964,14.803,-63.825,172.983,23.781,154.266
C07935=1071.971,15.083,-63.842,172.985,23.783,154.266
C07936=1071.977,15.333,-63.857,172.986,23.786,154.266
C07937=1071.983,15.582,-63.872,172.988,23.789,154.267
C07938=1071.989,15.832,-63.887,172.989,23.792,154.267
C07939=1071.995,16.082,-63.903,172.991,23.794,154.267
C07940=1072.000,16.331,-63.916,172.992,23.796,154.268
C07941=1072.007,16.581,-63.931,172.993,23.799,154.268
C07942=1072.013,16.830,-63.946,172.995,23.802,154.268
C07943=1072.018,17.080,-63.961,172.996,23.804,154.269
C07944=1072.024,17.329,-63.976,172.997,23.807,154.269
C07945=1072.030,17.578,-63.991,172.998,23.809,154.269
C07946=1072.036,17.828,-64.007,173.000,23.811,154.269
C07947=1072.042,18.077,-64.021,173.002,23.815,154.270
C07948=1072.048,18.327,-64.036,173.003,23.817,154.270
C07949=1072.054,18.576,-64.051,173.005,23.819,154.270
C07950=1072.060,18.826,-64.066,173.006,23.822,154.271
C07951=1072.066,19.076,-64.081,173.007,23.825,154.271
C07952=1072.074,19.439,-64.103,173.009,23.828,154.271
C07953=1072.083,19.803,-64.125,173.011,23.832,154.272
C07954=1072.092,20.168,-64.146,173.013,23.836,154.272
C07955=1072.100,20.532,-64.168,173.015,23.839,154.273
C07956=1072.106,20.782,-64.184,173.016,23.842,154.273
C07957=1072.112,21.031,-64.198,173.018,23.845,154.273
C07958=1072.118,21.281,-64.214,173.019,23.847,154.274
C07959=1072.124,21.530,-64.229,173.021,23.850,154.274
C07960=1072.130,21.779,-64.244,173.022,23.853,154.274
C07961=1072.136,22.029,-64.259,173.024,23.855,154.275
C07962=1072.142,22.278,-64.274,173.025,23.857,154.275
C07963=1072.147,22.528,-64.290,173.026,23.860,154.275
C07964=1072.153,22.777,-64.305,173.027,23.863,154.276
C07965=1072.159,23.027,-64.320,173.029,23.865,154.276
C07966=1072.165,23.276,-64.335,173.030,23.868,154.276
C07967=1072.171,23.526,-64.350,173.031,23.871,154.277
C07968=1072.177,23.775,-64.366,173.033,23.873,154.277
C07969=1072.183,24.024,-64.380,173.035,23.876,154.277
C07970=1072.189,24.274,-64.396,173.036,23.879,154.278
C07971=1072.195,24.524,-64.411,173.037,23.881,154.278
C07972=1072.200,24.773,-64.426,173.039,23.883,154.278
C07973=1072.206,25.023,-64.441,173.040,23.886,154.278
C07974=1072.213,25.272,-64.457,173.041,23.889,154.279
C07975=1072.218,25.521,-64.472,173.043,23.891,154.279
C07976=1072.225,25.771,-64.487,173.044,23.894,154.279
C07977=1072.230,26.021,-64.502,173.045,23.896,154.280
C07978=1072.237,26.270,-64.517,173.047,23.899,154.280
C07979=1072.242,26.519,-64.533,173.049,23.902,154.280
C07980=1072.248,26.769,-64.548,173.050,23.904,154.281
C07981=1072.254,27.018,-64.564,173.051,23.907,154.281
C07982=1072.260,27.267,-64.578,173.052,23.909,154.281
C07983=1072.266,27.517,-64.594,173.054,23.912,154.282
C07984=1072.272,27.766,-64.609,173.055,23.915,154.282
C07985=1072.278,28.016,-64.625,173.056,23.917,154.282
C07986=1072.284,28.265,-64.640,173.058,23.919,154.282
C07987=1072.289,28.515,-64.656,173.059,23.922,154.283
C07988=1072.296,28.764,-64.671,173.061,23.925,154.283
C07989=1072.302,29.014,-64.686,173.062,23.928,154.283
C07990=1072.307,29.263,-64.702,173.064,23.930,154.284
C07991=1072.313,29.513,-64.717,173.065,23.933,154.284
C07992=1072.323,29.930,-64.743,173.067,23.937,154.285
C07993=1072.332,30.346,-64.769,173.070,23.942,154.285
C07994=1072.342,30.763,-64.795,173.071,23.945,154.286
C07995=1072.352,31.180,-64.821,173.074,23.950,154.286
C07996=1072.358,31.430,-64.836,173.075,23.953,154.287
C07997=1072.364,31.680,-64.852,173.077,23.955,154.287
C07998=1072.370,31.929,-64.867,173.078,23.958,154.287
C07999=1072.375,32.178,-64.883,173.079,23.960,154.287
C08000=1072.381,32.427,-64.899,173.081,23.964,154.288
C08001=1072.388,32.677,-64.914,173.083,23.966,154.288
C08002=1072.394,32.926,-64.930,173.084,23.968,154.288
C08003=1072.399,33.176,-64.945,173.085,23.971,154.289
C08004=1072.405,33.425,-64.960,173.087,23.974,154.289
C08005=1072.411,33.675,-64.976,173.088,23.976,154.289
C08006=1072.417,33.925,-64.992,173.089,23.979,154.290
C08007=1072.423,34.174,-65.008,173.091,23.981,154.290
C08008=1072.428,34.423,-65.023,173.092,23.984,154.290
C08009=1072.434,34.672,-65.039,173.094,23.987,154.291
C08010=1072.440,34.922,-65.055,173.095,23.989,154.291
C08011=1072.447,35.171,-65.070,173.097,23.992,154.291
C08012=1072.452,35.421,-65.086,173.098,23.995,154.292
C08013=1072.458,35.671,-65.102,173.099,23.997,154.292
C08014=1072.464,35.920,-65.117,173.100,24.000,154.292
C08015=1072.470,36.169,-65.133,173.102,24.002,154.293
C08016=1072.476,36.419,-65.148,173.103,24.005,154.293
C08017=1072.482,36.668,-65.165,173.104,24.007,154.293
C08018=1072.488,36.917,-65.180,173.107,24.010,154.293
C08019=1072.494,37.167,-65.196,173.108,24.013,154.294
C08020=1072.500,37.417,-65.212,173.109,24.015,154.294
C08021=1072.506,37.666,-65.227,173.110,24.018,154.294
C08022=1072.512,37.915,-65.243,173.112,24.021,154.295
C08023=1072.517,38.165,-65.259,173.113,24.023,154.295
C08024=1072.523,38.414,-65.275,173.114,24.026,154.296
C08025=1072.529,38.664,-65.291,173.116,24.028,154.296
C08026=1072.535,38.914,-65.307,173.118,24.031,154.296
C08027=1072.540,39.162,-65.322,173.119,24.034,154.297
C08028=1072.546,39.411,-65.339,173.120,24.036,154.297
C08029=1072.553,39.661,-65.354,173.122,24.039,154.297
C08030=1072.559,39.911,-65.370,173.123,24.042,154.297
C08031=1072.564,40.160,-65.386,173.124,24.044,154.298
C08032=1072.570,40.410,-65.402,173.125,24.047,154.298
C08033=1072.576,40.659,-65.418,173.127,24.049,154.298
C08034=1072.581,40.908,-65.434,173.128,24.052,154.299
C08035=1072.587,41.158,-65.449,173.130,24.055,154.299
C08036=1072.593,41.407,-65.466,173.132,24.057,154.299
C08037=1072.599,41.656,-65.482,173.133,24.060,154.300
C08038=1072.605,41.906,-65.497,173.134,24.063,154.300
C08039=1072.611,42.156,-65.514,173.135,24.065,154.300
C08040=1072.617,42.405,-65.529,173.137,24.068,154.301
C08041=1072.623,42.654,-65.546,173.138,24.071,154.301
C08042=1072.628,42.903,-65.561,173.139,24.073,154.301
C08043=1072.634,43.153,-65.577,173.141,24.076,154.302
C08044=1072.640,43.402,-65.593,173.143,24.079,154.302
C08045=1072.646,43.651,-65.610,173.144,24.081,154.302
C08046=1072.652,43.901,-65.625,173.145,24.084,154.303
C08047=1072.658,44.151,-65.641,173.147,24.086,154.303
C08048=1072.664,44.400,-65.658,173.148,24.089,154.303
C08049=1072.670,44.650,-65.674,173.149,24.092,154.304
C08050=1072.675,44.899,-65.691,173.150,24.094,154.304
C08051=1072.680,45.148,-65.706,173.153,24.097,154.304
C08052=1072.686,45.398,-65.722,173.154,24.100,154.305
C08053=1072.692,45.647,-65.738,173.155,24.103,154.305
C08054=1072.698,45.896,-65.755,173.156,24.105,154.305
C08055=1072.704,46.146,-65.771,173.158,24.108,154.306
C08056=1072.710,46.428,-65.789,173.160,24.111,154.306
C08057=1072.716,46.711,-65.808,173.161,24.114,154.306
C08058=1072.723,46.992,-65.826,173.162,24.117,154.307
C08059=1072.730,47.275,-65.844,173.164,24.120,154.307
C08060=1072.735,47.524,-65.861,173.166,24.123,154.308
C08061=1072.741,47.774,-65.877,173.167,24.125,154.308
C08062=1072.747,48.023,-65.893,173.168,24.128,154.308
C08063=1072.752,48.272,-65.910,173.170,24.130,154.309
C08064=1072.758,48.521,-65.926,173.171,24.133,154.309
C08065=1072.764,48.771,-65.942,173.173,24.136,154.309
C08066=1072.770,49.020,-65.958,173.174,24.139,154.310
C08067=1072.776,49.269,-65.975,173.176,24.141,154.310
C08068=1072.782,49.519,-65.991,173.177,24.144,154.310
C08069=1072.787,49.768,-66.008,173.178,24.147,154.311
C08070=1072.793,50.018,-66.024,173.179,24.149,154.311
C08071=1072.799,50.267,-66.040,173.181,24.152,154.311
C08072=1072.805,50.517,-66.056,173.182,24.154,154.312
C08073=1072.811,50.766,-66.073,173.184,24.158,154.312
C08074=1072.816,51.015,-66.090,173.186,24.160,154.312
C08075=1072.822,51.265,-66.106,173.187,24.162,154.312
C08076=1072.828,51.514,-66.122,173.188,24.165,154.313
C08077=1072.834,51.763,-66.138,173.189,24.168,154.313
C08078=1072.840,52.013,-66.155,173.191,24.171,154.314
C08079=1072.845,52.262,-66.171,173.192,24.173,154.314
C08080=1072.851,52.512,-66.188,173.194,24.176,154.314
C08081=1072.857,52.761,-66.204,173.195,24.179,154.315
C08082=1072.863,53.010,-66.220,173.197,24.181,154.315
C08083=1072.869,53.260,-66.236,173.198,24.184,154.315
C08084=1072.874,53.509,-66.253,173.199,24.186,154.316
C08085=1072.880,53.759,-66.270,173.201,24.189,154.316
C08086=1072.886,54.008,-66.286,173.202,24.192,154.316
C08087=1072.892,54.257,-66.302,173.204,24.194,154.316
C08088=1072.897,54.507,-66.319,173.205,24.197,154.317
C08089=1072.904,54.757,-66.336,173.207,24.200,154.317
C08090=1072.910,55.006,-66.353,173.208,24.202,154.317
C08091=1072.916,55.255,-66.369,173.209,24.205,154.318
C08092=1072.921,55.505,-66.386,173.211,24.207,154.318
C08093=1072.927,55.754,-66.402,173.212,24.210,154.318
C08094=1072.933,56.004,-66.418,173.214,24.213,154.319
C08095=1072.939,56.252,-66.435,173.215,24.215,154.319
C08096=1072.944,56.502,-66.452,173.217,24.218,154.319
C08097=1072.950,56.751,-66.468,173.218,24.221,154.320
C08098=1072.956,57.001,-66.484,173.219,24.223,154.320
C08099=1072.962,57.250,-66.501,173.221,24.226,154.320
C08100=1072.968,57.500,-66.519,173.222,24.228,154.321
C08101=1072.974,57.749,-66.535,173.224,24.231,154.321
C08102=1072.980,57.998,-66.551,173.225,24.234,154.321
C08103=1072.986,58.248,-66.567,173.227,24.236,154.322
C08104=1072.992,58.497,-66.585,173.228,24.239,154.322
C08105=1072.998,58.746,-66.601,173.229,24.242,154.322
C08106=1073.004,58.996,-66.618,173.231,24.244,154.323
C08107=1073.009,59.245,-66.634,173.232,24.246,154.323
C08108=1073.016,59.495,-66.652,173.234,24.250,154.323
C08109=1073.022,59.744,-66.668,173.236,24.252,154.324
C08110=1073.028,59.993,-66.684,173.237,24.254,154.324
C08111=1073.033,60.243,-66.701,173.238,24.257,154.324
C08112=1073.039,60.492,-66.718,173.240,24.260,154.325
C08113=1073.045,60.741,-66.734,173.241,24.262,154.325
C08114=1073.051,60.991,-66.752,173.243,24.265,154.325
C08115=1073.057,61.240,-66.768,173.244,24.268,154.326
C08116=1073.063,61.490,-66.785,173.246,24.270,154.326
C08117=1073.068,61.739,-66.802,173.247,24.273,154.326
C08118=1073.075,61.988,-66.819,173.248,24.275,154.327
C08119=1073.081,62.238,-66.835,173.250,24.278,154.327
C08120=1073.087,62.519,-66.855,173.252,24.281,154.327
C08121=1073.094,62.801,-66.874,173.253,24.284,154.328
C08122=1073.102,63.083,-66.893,173.255,24.287,154.328
C08123=1073.108,63.365,-66.911,173.256,24.289,154.328
C08124=1073.113,63.614,-66.928,173.258,24.292,154.329
C08125=1073.120,63.864,-66.945,173.259,24.295,154.329
C08126=1073.125,64.113,-66.962,173.261,24.297,154.329
C08127=1073.131,64.363,-66.979,173.263,24.300,154.329
C08128=1073.138,64.611,-66.996,173.264,24.303,154.330
C08129=1073.143,64.861,-67.013,173.265,24.305,154.330
C08130=1073.149,65.111,-67.029,173.267,24.308,154.330
C08131=1073.155,65.360,-67.047,173.268,24.310,154.331
C08132=1073.160,65.610,-67.064,173.270,24.313,154.331
C08133=1073.166,65.858,-67.081,173.271,24.316,154.332
C08134=1073.172,66.108,-67.097,173.273,24.318,154.332
C08135=1073.179,66.358,-67.115,173.274,24.321,154.332
C08136=1073.184,66.607,-67.132,173.275,24.324,154.332
C08137=1073.190,66.856,-67.149,173.277,24.326,154.333
C08138=1073.196,67.105,-67.166,173.279,24.329,154.333
C08139=1073.202,67.355,-67.183,173.280,24.332,154.333
C08140=1073.208,67.604,-67.200,173.281,24.334,154.334
C08141=1073.213,67.854,-67.217,173.283,24.337,154.334
C08142=1073.219,68.102,-67.234,173.284,24.339,154.334
C08143=1073.225,68.353,-67.251,173.285,24.342,154.335
C08144=1073.231,68.602,-67.268,173.288,24.345,154.335
C08145=1073.236,68.851,-67.285,173.289,24.347,154.335
C08146=1073.242,69.100,-67.303,173.290,24.350,154.336
C08147=1073.248,69.349,-67.320,173.292,24.353,154.336
C08148=1073.254,69.599,-67.337,173.293,24.355,154.336
C08149=1073.260,69.848,-67.354,173.294,24.358,154.337
C08150=1073.266,70.097,-67.371,173.296,24.361,154.337
C08151=1073.272,70.347,-67.389,173.298,24.364,154.337
C08152=1073.277,70.597,-67.406,173.299,24.366,154.338
C08153=1073.283,70.846,-67.423,173.300,24.368,154.338
C08154=1073.289,71.095,-67.440,173.302,24.371,154.338
C08155=1073.295,71.345,-67.458,173.303,24.374,154.339
C08156=1073.301,71.594,-67.474,173.305,24.377,154.339
C08157=1073.306,71.843,-67.492,173.306,24.379,154.339
C08158=1073.312,72.092,-67.509,173.308,24.381,154.340
C08159=1073.318,72.342,-67.527,173.309,24.384,154.340
C08160=1073.324,72.591,-67.544,173.310,24.387,154.340
C08161=1073.329,72.840,-67.561,173.312,24.389,154.341
C08162=1073.335,73.089,-67.579,173.314,24.392,154.341
C08163=1073.341,73.340,-67.596,173.315,24.395,154.341
C08164=1073.347,73.588,-67.613,173.316,24.398,154.342
C08165=1073.352,73.837,-67.630,173.318,24.400,154.342
C08166=1073.358,74.087,-67.648,173.319,24.402,154.342
C08167=1073.364,74.336,-67.666,173.321,24.406,154.343
C08168=1073.370,74.586,-67.682,173.323,24.408,154.343
C08169=1073.376,74.835,-67.700,173.324,24.411,154.343
C08170=1073.382,75.084,-67.718,173.325,24.413,154.344
C08171=1073.387,75.333,-67.735,173.327,24.416,154.344
C08172=1073.393,75.583,-67.753,173.329,24.419,154.344
C08173=1073.399,75.832,-67.770,173.330,24.421,154.345
C08174=1073.405,76.081,-67.787,173.332,24.424,154.345
C08175=1073.411,76.331,-67.805,173.333,24.427,154.345
C08176=1073.416,76.580,-67.823,173.334,24.429,154.346
C08177=1073.422,76.829,-67.840,173.336,24.431,154.346
C08178=1073.429,77.079,-67.857,173.338,24.434,154.346
C08179=1073.434,77.328,-67.874,173.339,24.437,154.346
C08180=1073.439,77.577,-67.892,173.340,24.439,154.347
C08181=1073.446,77.827,-67.910,173.342,24.442,154.347
C08182=1073.451,78.076,-67.927,173.343,24.444,154.347
C08183=1073.457,78.325,-67.945,173.345,24.448,154.348
C08184=1073.463,78.607,-67.965,173.347,24.450,154.348
C08185=1073.470,78.889,-67.985,173.349,24.453,154.349
C08186=1073.476,79.171,-68.005,173.350,24.456,154.349
C08187=1073.483,79.452,-68.025,173.352,24.459,154.349
C08188=1073.489,79.702,-68.043,173.353,24.462,154.350
C08189=1073.494,79.951,-68.060,173.355,24.465,154.350
C08190=1073.500,80.200,-68.078,173.356,24.467,154.350
C08191=1073.506,80.450,-68.096,173.357,24.470,154.351
C08192=1073.511,80.699,-68.113,173.360,24.473,154.351
C08193=1073.518,80.949,-68.131,173.361,24.475,154.351
C08194=1073.523,81.198,-68.149,173.362,24.478,154.352
C08195=1073.529,81.447,-68.166,173.364,24.480,154.352
C08196=1073.535,81.696,-68.184,173.365,24.483,154.352
C08197=1073.540,81.945,-68.202,173.367,24.486,154.353
C08198=1073.546,82.194,-68.219,173.368,24.488,154.353
C08199=1073.552,82.444,-68.237,173.370,24.491,154.353
C08200=1073.557,82.693,-68.255,173.371,24.494,154.354
C08201=1073.564,82.943,-68.273,173.372,24.496,154.354
C08202=1073.569,83.192,-68.290,173.375,24.499,154.354
C08203=1073.575,83.442,-68.308,173.376,24.502,154.355
C08204=1073.581,83.691,-68.326,173.377,24.504,154.355
C08205=1073.586,83.940,-68.344,173.379,24.507,154.355
C08206=1073.592,84.190,-68.361,173.380,24.509,154.356
C08207=1073.598,84.439,-68.379,173.382,24.512,154.356
C08208=1073.604,84.688,-68.397,173.383,24.515,154.356
C08209=1073.610,84.937,-68.415,173.385,24.517,154.356
C08210=1073.616,85.186,-68.433,173.386,24.520,154.357
C08211=1073.621,85.436,-68.451,173.387,24.522,154.357
C08212=1073.626,85.685,-68.469,173.390,24.526,154.358
C08213=1073.632,85.935,-68.487,173.391,24.528,154.358
C08214=1073.638,86.184,-68.504,173.392,24.530,154.358
C08215=1073.644,86.433,-68.523,173.394,24.533,154.359
C08216=1073.650,86.682,-68.541,173.396,24.536,154.359
C08217=1073.656,86.932,-68.559,173.397,24.538,154.359
C08218=1073.661,87.181,-68.576,173.398,24.541,154.359
C08219=1073.668,87.430,-68.594,173.400,24.543,154.360
C08220=1073.673,87.679,-68.612,173.401,24.546,154.360
C08221=1073.679,87.929,-68.630,173.404,24.549,154.360
C08222=1073.685,88.178,-68.648,173.405,24.551,154.361
C08223=1073.690,88.428,-68.666,173.406,24.554,154.361
C08224=1073.696,88.676,-68.685,173.408,24.556,154.361
C08225=1073.702,88.926,-68.703,173.409,24.559,154.362
C08226=1073.708,89.175,-68.720,173.411,24.562,154.362
C08227=1073.714,89.425,-68.738,173.412,24.564,154.362
C08228=1073.720,89.674,-68.757,173.414,24.567,154.363
C08229=1073.726,89.923,-68.774,173.415,24.569,154.363
C08230=1073.732,90.172,-68.792,173.417,24.572,154.363
C08231=1073.738,90.421,-68.811,173.419,24.574,154.363
C08232=1073.743,90.671,-68.829,173.420,24.577,154.364
C08233=1073.749,90.920,-68.847,173.421,24.580,154.364
C08234=1073.755,91.170,-68.865,173.424,24.582,154.364
C08235=1073.761,91.418,-68.883,173.425,24.585,154.365
C08236=1073.766,91.668,-68.901,173.426,24.588,154.365
C08237=1073.772,91.917,-68.920,173.428,24.590,154.366
C08238=1073.778,92.166,-68.938,173.429,24.593,154.366
C08239=1073.783,92.416,-68.956,173.431,24.595,154.366
C08240=1073.789,92.665,-68.974,173.432,24.598,154.366
C08241=1073.795,92.914,-68.992,173.434,24.601,154.367
C08242=1073.800,93.163,-69.011,173.435,24.603,154.367
C08243=1073.807,93.413,-69.029,173.437,24.606,154.367
C08244=1073.812,93.662,-69.047,173.439,24.609,154.368
C08245=1073.818,93.911,-69.066,173.440,24.611,154.368
C08246=1073.823,94.161,-69.084,173.441,24.614,154.368
C08247=1073.830,94.410,-69.102,173.444,24.617,154.369
C08248=1073.836,94.692,-69.123,173.445,24.619,154.369
C08249=1073.843,94.973,-69.144,173.447,24.623,154.369
C08250=1073.849,95.255,-69.165,173.449,24.625,154.370
C08251=1073.855,95.537,-69.186,173.451,24.628,154.370
C08252=1073.861,95.787,-69.203,173.452,24.631,154.371
C08253=1073.867,96.035,-69.222,173.453,24.634,154.371
C08254=1073.872,96.285,-69.240,173.455,24.636,154.371
C08255=1073.878,96.534,-69.259,173.457,24.639,154.371
C08256=1073.884,96.783,-69.277,173.458,24.641,154.372
C08257=1073.890,97.033,-69.296,173.460,24.644,154.372
C08258=1073.895,97.282,-69.313,173.461,24.646,154.372
C08259=1073.901,97.531,-69.333,173.463,24.649,154.373
C08260=1073.907,97.780,-69.350,173.465,24.652,154.373
C08261=1073.913,98.029,-69.369,173.466,24.654,154.373
C08262=1073.919,98.279,-69.388,173.467,24.657,154.374
C08263=1073.924,98.528,-69.406,173.470,24.660,154.374
C08264=1073.930,98.777,-69.425,173.471,24.662,154.374
C08265=1073.936,99.027,-69.443,173.472,24.664,154.375
C08266=1073.942,99.275,-69.461,173.474,24.668,154.375
C08267=1073.947,99.525,-69.480,173.476,24.670,154.375
C08268=1073.954,99.775,-69.498,173.477,24.672,154.375
C08269=1073.959,100.023,-69.517,173.479,24.675,154.376
C08270=1073.965,100.273,-69.536,173.481,24.678,154.376
C08271=1073.970,100.523,-69.554,173.482,24.680,154.376
C08272=1073.976,100.771,-69.573,173.484,24.683,154.377
C08273=1073.983,101.020,-69.591,173.485,24.685,154.377
C08274=1073.988,101.270,-69.610,173.487,24.688,154.377
C08275=1073.994,101.519,-69.628,173.489,24.690,154.378
C08276=1074.000,101.768,-69.647,173.490,24.693,154.378
C08277=1074.005,102.018,-69.666,173.491,24.696,154.378
C08278=1074.011,102.266,-69.684,173.493,24.698,154.379
C08279=1074.017,102.516,-69.703,173.495,24.701,154.379
C08280=1074.022,102.765,-69.723,173.496,24.704,154.379
C08281=1074.028,103.014,-69.740,173.498,24.706,154.380
C08282=1074.033,103.264,-69.759,173.500,24.709,154.380
C08283=1074.040,103.513,-69.778,173.501,24.712,154.380
C08284=1074.045,103.762,-69.797,173.502,24.714,154.381
C08285=1074.050,104.012,-69.815,173.505,24.717,154.381
C08286=1074.057,104.261,-69.834,173.506,24.719,154.381
C08287=1074.062,104.510,-69.853,173.507,24.722,154.382
C08288=1074.068,104.759,-69.872,173.509,24.724,154.382
C08289=1074.074,105.008,-69.891,173.511,24.727,154.382
C08290=1074.079,105.258,-69.909,173.512,24.730,154.382
C08291=1074.084,105.507,-69.928,173.514,24.732,154.383
C08292=1074.091,105.756,-69.947,173.516,24.735,154.383
C08293=1074.097,106.005,-69.966,173.517,24.738,154.383
C08294=1074.102,106.254,-69.985,173.519,24.740,154.384
C08295=1074.108,106.503,-70.004,173.520,24.742,154.384
C08296=1074.114,106.753,-70.023,173.522,24.745,154.384
C08297=1074.118,107.002,-70.041,173.524,24.748,154.385
C08298=1074.125,107.251,-70.060,173.525,24.750,154.385
C08299=1074.131,107.501,-70.079,173.527,24.753,154.385
C08300=1074.136,107.750,-70.098,173.529,24.756,154.386
C08301=1074.142,107.999,-70.116,173.530,24.758,154.386
C08302=1074.148,108.248,-70.136,173.531,24.760,154.386
C08303=1074.153,108.497,-70.155,173.534,24.764,154.387
C08304=1074.160,108.747,-70.174,173.535,24.766,154.387
C08305=1074.166,108.996,-70.193,173.536,24.768,154.387
C08306=1074.171,109.245,-70.212,173.539,24.771,154.387
C08307=1074.176,109.494,-70.231,173.540,24.774,154.388
C08308=1074.183,109.743,-70.250,173.541,24.776,154.388
C08309=1074.189,109.993,-70.269,173.543,24.779,154.388
C08310=1074.194,110.242,-70.288,173.545,24.781,154.389
C08311=1074.200,110.491,-70.306,173.546,24.784,154.389
C08312=1074.207,110.773,-70.328,173.549,24.787,154.389
C08313=1074.213,111.054,-70.349,173.550,24.790,154.390
C08314=1074.220,111.336,-70.372,173.552,24.792,154.390
C08315=1074.226,111.618,-70.393,173.554,24.796,154.390
C08316=1074.232,111.868,-70.412,173.556,24.798,154.391
C08317=1074.238,112.117,-70.431,173.557,24.801,154.391
C08318=1074.243,112.366,-70.450,173.558,24.803,154.391
C08319=1074.248,112.615,-70.469,173.561,24.806,154.392
C08320=1074.254,112.865,-70.488,173.562,24.808,154.392
C08321=1074.261,113.113,-70.508,173.563,24.811,154.392
C08322=1074.266,113.363,-70.527,173.566,24.814,154.393
C08323=1074.272,113.612,-70.546,173.567,24.816,154.393
C08324=1074.277,113.861,-70.565,173.569,24.818,154.393
C08325=1074.283,114.110,-70.584,173.571,24.822,154.394
C08326=1074.289,114.360,-70.604,173.572,24.824,154.394
C08327=1074.294,114.609,-70.623,173.574,24.826,154.394
C08328=1074.300,114.858,-70.643,173.576,24.829,154.394
C08329=1074.306,115.107,-70.662,173.577,24.832,154.395
C08330=1074.311,115.356,-70.681,173.579,24.834,154.395
C08331=1074.317,115.606,-70.700,173.581,24.837,154.395
C08332=1074.322,115.855,-70.719,173.582,24.840,154.396
C08333=1074.328,116.104,-70.739,173.584,24.842,154.396
C08334=1074.334,116.353,-70.759,173.586,24.845,154.396
C08335=1074.339,116.602,-70.778,173.587,24.848,154.397
C08336=1074.345,116.851,-70.797,173.589,24.850,154.397
C08337=1074.351,117.100,-70.817,173.591,24.853,154.397
C08338=1074.357,117.350,-70.836,173.592,24.855,154.398
C08339=1074.362,117.599,-70.855,173.594,24.858,154.398
C08340=1074.367,117.849,-70.875,173.595,24.860,154.398
C08341=1074.373,118.097,-70.895,173.597,24.863,154.399
C08342=1074.378,118.346,-70.914,173.598,24.866,154.399
C08343=1074.384,118.596,-70.933,173.600,24.868,154.399
C08344=1074.390,118.845,-70.953,173.602,24.871,154.399
C08345=1074.396,119.094,-70.972,173.603,24.873,154.400
C08346=1074.401,119.344,-70.992,173.606,24.876,154.400
C08347=1074.407,119.593,-71.011,173.607,24.878,154.400
C08348=1074.413,119.842,-71.031,173.609,24.881,154.401
C08349=1074.418,120.091,-71.050,173.611,24.884,154.401
C08350=1074.424,120.339,-71.070,173.612,24.886,154.401
C08351=1074.429,120.589,-71.089,173.614,24.889,154.402
C08352=1074.435,120.838,-71.109,173.616,24.891,154.402
C08353=1074.441,121.087,-71.129,173.617,24.894,154.402
C08354=1074.446,121.337,-71.148,173.619,24.897,154.403
C08355=1074.452,121.586,-71.168,173.621,24.899,154.403
C08356=1074.458,121.835,-71.187,173.622,24.902,154.403
C08357=1074.464,122.084,-71.206,173.624,24.904,154.404
C08358=1074.470,122.333,-71.226,173.626,24.907,154.404
C08359=1074.475,122.583,-71.246,173.627,24.909,154.404
C08360=1074.481,122.832,-71.266,173.629,24.912,154.404
C08361=1074.486,123.081,-71.285,173.631,24.915,154.405
C08362=1074.492,123.330,-71.305,173.632,24.917,154.405
C08363=1074.498,123.579,-71.325,173.634,24.920,154.405
C08364=1074.503,123.828,-71.344,173.636,24.922,154.406
C08365=1074.508,124.077,-71.364,173.638,24.925,154.406
C08366=1074.514,124.326,-71.384,173.640,24.928,154.406
C08367=1074.520,124.576,-71.403,173.641,24.930,154.407
C08368=1074.526,124.824,-71.423,173.643,24.932,154.407
C08369=1074.532,125.074,-71.442,173.645,24.935,154.407
C08370=1074.538,125.323,-71.462,173.646,24.937,154.407
C08371=1074.543,125.572,-71.482,173.648,24.940,154.408
C08372=1074.549,125.821,-71.502,173.650,24.943,154.408
C08373=1074.554,126.071,-71.521,173.651,24.945,154.408
C08374=1074.561,126.320,-71.542,173.653,24.948,154.409
C08375=1074.567,126.569,-71.562,173.655,24.950,154.409
C08376=1074.573,126.851,-71.584,173.657,24.953,154.409
C08377=1074.580,127.133,-71.606,173.659,24.956,154.410
C08378=1074.586,127.415,-71.629,173.661,24.959,154.410
C08379=1074.592,127.696,-71.650,173.663,24.962,154.410
C08380=1074.598,127.945,-71.670,173.665,24.964,154.410
C08381=1074.604,128.194,-71.691,173.666,24.967,154.411
C08382=1074.610,128.444,-71.711,173.668,24.970,154.411
C08383=1074.616,128.693,-71.731,173.670,24.972,154.411
C08384=1074.622,128.942,-71.750,173.672,24.975,154.412
C08385=1074.627,129.192,-71.770,173.673,24.977,154.412
C08386=1074.633,129.440,-71.790,173.675,24.979,154.412
C08387=1074.639,129.689,-71.810,173.677,24.982,154.413
C08388=1074.645,129.938,-71.830,173.678,24.984,154.413
C08389=1074.650,130.187,-71.849,173.681,24.987,154.413
C08390=1074.656,130.437,-71.870,173.682,24.990,154.413
C08391=1074.662,130.685,-71.890,173.684,24.992,154.414
C08392=1074.668,130.936,-71.910,173.686,24.995,154.414
C08393=1074.674,131.184,-71.930,173.687,24.997,154.414
C08394=1074.679,131.433,-71.950,173.690,25.000,154.415
C08395=1074.685,131.682,-71.970,173.691,25.002,154.415
C08396=1074.691,131.931,-71.990,173.692,25.004,154.415
C08397=1074.696,132.181,-72.010,173.695,25.007,154.415
C08398=1074.702,132.430,-72.030,173.696,25.009,154.416
C08399=1074.708,132.678,-72.050,173.698,25.012,154.416
C08400=1074.713,132.928,-72.070,173.700,25.015,154.416
C08401=1074.720,133.177,-72.091,173.701,25.017,154.417
C08402=1074.725,133.427,-72.110,173.704,25.020,154.417
C08403=1074.731,133.676,-72.130,173.705,25.022,154.417
C08404=1074.736,133.925,-72.151,173.707,25.025,154.418
C08405=1074.742,134.174,-72.171,173.709,25.028,154.418
C08406=1074.747,134.423,-72.191,173.710,25.030,154.418
C08407=1074.753,134.672,-72.211,173.712,25.033,154.418
C08408=1074.759,134.921,-72.232,173.714,25.035,154.419
C08409=1074.765,135.169,-72.252,173.716,25.038,154.419
C08410=1074.771,135.419,-72.273,173.717,25.040,154.419
C08411=1074.776,135.669,-72.292,173.719,25.043,154.420
C08412=1074.782,135.918,-72.313,173.721,25.045,154.420
C08413=1074.788,136.167,-72.333,173.723,25.048,154.420
C08414=1074.793,136.416,-72.353,173.725,25.050,154.420
C08415=1074.799,136.665,-72.373,173.726,25.053,154.421
C08416=1074.804,136.914,-72.394,173.729,25.055,154.421
C08417=1074.811,137.163,-72.414,173.730,25.058,154.421
C08418=1074.816,137.412,-72.435,173.731,25.060,154.422
C08419=1074.822,137.661,-72.455,173.734,25.063,154.422
C08420=1074.827,137.910,-72.475,173.735,25.065,154.422
C08421=1074.832,138.159,-72.496,173.737,25.068,154.423
C08422=1074.839,138.409,-72.516,173.739,25.070,154.423
C08423=1074.844,138.658,-72.537,173.741,25.073,154.423
C08424=1074.850,138.907,-72.556,173.742,25.076,154.423
C08425=1074.855,139.156,-72.577,173.745,25.079,154.424
C08426=1074.861,139.405,-72.598,173.746,25.081,154.424
C08427=1074.868,139.654,-72.619,173.748,25.083,154.424
C08428=1074.873,139.903,-72.639,173.750,25.086,154.425
C08429=1074.879,140.152,-72.659,173.751,25.088,154.425
C08430=1074.884,140.401,-72.680,173.754,25.091,154.425
C08431=1074.889,140.650,-72.700,173.755,25.093,154.425
C08432=1074.896,140.900,-72.721,173.757,25.096,154.426
C08433=1074.901,141.149,-72.741,173.759,25.099,154.426
C08434=1074.907,141.398,-72.762,173.761,25.101,154.426
C08435=1074.912,141.646,-72.783,173.763,25.104,154.427
C08436=1074.918,141.895,-72.803,173.764,25.106,154.427
C08437=1074.924,142.145,-72.824,173.766,25.109,154.427
C08438=1074.929,142.394,-72.844,173.768,25.111,154.428
C08439=1074.934,142.643,-72.865,173.770,25.114,154.428
C08440=1074.941,142.925,-72.888,173.772,25.117,154.428
C08441=1074.948,143.207,-72.912,173.774,25.120,154.429
C08442=1074.954,143.488,-72.935,173.776,25.122,154.429
C08443=1074.961,143.770,-72.958,173.778,25.125,154.429
C08444=1074.966,144.019,-72.979,173.780,25.128,154.429
C08445=1074.972,144.268,-72.999,173.782,25.130,154.430
C08446=1074.978,144.517,-73.020,173.783,25.133,154.430
C08447=1074.983,144.766,-73.041,173.786,25.136,154.430
C08448=1074.989,145.015,-73.062,173.787,25.138,154.431
C08449=1074.994,145.264,-73.083,173.789,25.141,154.431
C08450=1075.001,145.514,-73.103,173.791,25.143,154.431
C08451=1075.006,145.763,-73.124,173.793,25.146,154.431
C08452=1075.011,146.012,-73.144,173.795,25.148,154.432
C08453=1075.017,146.260,-73.166,173.797,25.151,154.432
C08454=1075.023,146.510,-73.186,173.798,25.153,154.432
C08455=1075.029,146.758,-73.207,173.801,25.156,154.433
C08456=1075.034,147.007,-73.228,173.802,25.158,154.433
C08457=1075.040,147.257,-73.249,173.804,25.161,154.433
C08458=1075.046,147.506,-73.270,173.806,25.163,154.434
C08459=1075.052,147.755,-73.290,173.808,25.166,154.434
C08460=1075.058,148.004,-73.311,173.810,25.168,154.434
C08461=1075.063,148.253,-73.332,173.812,25.171,154.434
C08462=1075.068,148.502,-73.353,173.813,25.173,154.435
C08463=1075.075,148.751,-73.374,173.816,25.176,154.435
C08464=1075.080,149.000,-73.395,173.817,25.178,154.435
C08465=1075.085,149.249,-73.416,173.819,25.181,154.435
C08466=1075.091,149.499,-73.437,173.821,25.184,154.436
C08467=1075.096,149.748,-73.458,173.823,25.186,154.436
C08468=1075.102,149.996,-73.479,173.824,25.189,154.436
C08469=1075.108,150.246,-73.500,173.827,25.191,154.437
C08470=1075.113,150.495,-73.521,173.828,25.194,154.437
C08471=1075.119,150.744,-73.542,173.831,25.196,154.437
C08472=1075.125,150.993,-73.563,173.832,25.199,154.438
C08473=1075.130,151.242,-73.584,173.834,25.201,154.438
C08474=1075.136,151.491,-73.606,173.836,25.204,154.438
C08475=1075.142,151.740,-73.627,173.838,25.207,154.438
C08476=1075.147,151.989,-73.647,173.839,25.209,154.439
C08477=1075.153,152.238,-73.669,173.842,25.212,154.439
C08478=1075.158,152.487,-73.690,173.843,25.214,154.439
C08479=1075.164,152.736,-73.711,173.846,25.217,154.440
C08480=1075.170,152.986,-73.732,173.847,25.219,154.440
C08481=1075.175,153.234,-73.753,173.849,25.222,154.440
C08482=1075.182,153.483,-73.775,173.851,25.224,154.441
C08483=1075.187,153.732,-73.795,173.853,25.227,154.441
C08484=1075.192,153.981,-73.816,173.854,25.229,154.441
C08485=1075.198,154.231,-73.837,173.857,25.232,154.441
C08486=1075.204,154.479,-73.859,173.859,25.235,154.442
C08487=1075.210,154.728,-73.880,173.861,25.237,154.442
C08488=1075.215,154.978,-73.901,173.863,25.240,154.442
C08489=1075.221,155.227,-73.922,173.864,25.242,154.442
C08490=1075.227,155.475,-73.944,173.867,25.245,154.443
C08491=1075.233,155.724,-73.965,173.868,25.247,154.443
C08492=1075.238,155.974,-73.986,173.871,25.250,154.443
C08493=1075.243,156.222,-74.008,173.872,25.252,154.444
C08494=1075.249,156.472,-74.029,173.874,25.255,154.444
C08495=1075.255,156.721,-74.050,173.876,25.257,154.444
C08496=1075.261,156.970,-74.072,173.878,25.260,154.444
C08497=1075.266,157.218,-74.093,173.880,25.263,154.445
C08498=1075.272,157.467,-74.114,173.882,25.265,154.445
C08499=1075.277,157.716,-74.136,173.884,25.268,154.445
C08500=1075.283,157.966,-74.157,173.886,25.270,154.446
C08501=1075.289,158.215,-74.179,173.888,25.272,154.446
C08502=1075.294,158.463,-74.200,173.889,25.275,154.446
C08503=1075.301,158.713,-74.221,173.892,25.278,154.446
C08504=1075.306,158.995,-74.245,173.894,25.281,154.447
C08505=1075.313,159.276,-74.270,173.896,25.284,154.447
C08506=1075.319,159.557,-74.294,173.899,25.286,154.447
C08507=1075.325,159.838,-74.319,173.900,25.289,154.448
C08508=1075.331,160.088,-74.340,173.902,25.292,154.448
C08509=1075.337,160.337,-74.361,173.905,25.294,154.448
C08510=1075.343,160.586,-74.383,173.906,25.297,154.449
C08511=1075.349,160.834,-74.404,173.908,25.299,154.449
C08512=1075.354,161.084,-74.426,173.910,25.302,154.449
C08513=1075.360,161.332,-74.448,173.912,25.304,154.449
C08514=1075.366,161.582,-74.469,173.915,25.307,154.450
C08515=1075.371,161.830,-74.491,173.916,25.309,154.450
C08516=1075.377,162.080,-74.513,173.918,25.312,154.450
C08517=1075.382,162.328,-74.535,173.920,25.315,154.451
C08518=1075.387,162.577,-74.556,173.922,25.317,154.451
C08519=1075.393,162.826,-74.578,173.923,25.320,154.451
C08520=1075.398,163.075,-74.599,173.926,25.323,154.452
C08521=1075.404,163.324,-74.622,173.928,25.325,154.452
C08522=1075.409,163.573,-74.643,173.929,25.328,154.452
C08523=1075.415,163.822,-74.665,173.932,25.330,154.452
C08524=1075.420,164.071,-74.686,173.933,25.333,154.453
C08525=1075.426,164.320,-74.709,173.935,25.336,154.453
C08526=1075.430,164.569,-74.730,173.938,25.338,154.453
C08527=1075.437,164.819,-74.752,173.939,25.341,154.454
C08528=1075.441,165.067,-74.774,173.942,25.343,154.454
C08529=1075.448,165.317,-74.796,173.943,25.346,154.454
C08530=1075.452,165.565,-74.817,173.945,25.349,154.455
C08531=1075.459,165.815,-74.839,173.948,25.352,154.455
C08532=1075.464,166.063,-74.862,173.949,25.354,154.455
C08533=1075.470,166.312,-74.883,173.951,25.356,154.455
C08534=1075.475,166.561,-74.905,173.953,25.359,154.456
C08535=1075.480,166.810,-74.927,173.955,25.362,154.456
C08536=1075.486,167.060,-74.949,173.958,25.365,154.456
C08537=1075.491,167.308,-74.971,173.959,25.367,154.457
C08538=1075.498,167.557,-74.993,173.961,25.369,154.457
C08539=1075.502,167.806,-75.015,173.964,25.372,154.457
C08540=1075.508,168.055,-75.037,173.965,25.375,154.458
C08541=1075.514,168.304,-75.059,173.967,25.378,154.458
C08542=1075.519,168.553,-75.081,173.969,25.380,154.458
C08543=1075.525,168.802,-75.103,173.971,25.382,154.458
C08544=1075.530,169.051,-75.125,173.974,25.385,154.459
C08545=1075.536,169.300,-75.147,173.975,25.387,154.459
C08546=1075.542,169.549,-75.169,173.977,25.390,154.459
C08547=1075.547,169.798,-75.191,173.980,25.393,154.460
C08548=1075.553,170.047,-75.213,173.981,25.395,154.460
C08549=1075.558,170.296,-75.235,173.983,25.398,154.460
C08550=1075.564,170.545,-75.257,173.986,25.401,154.460
C08551=1075.570,170.794,-75.280,173.987,25.403,154.461
C08552=1075.574,171.043,-75.301,173.990,25.406,154.461
C08553=1075.581,171.292,-75.323,173.991,25.408,154.461
C08554=1075.586,171.541,-75.346,173.993,25.411,154.462
C08555=1075.591,171.789,-75.368,173.996,25.414,154.462
C08556=1075.598,172.038,-75.390,173.997,25.416,154.462
C08557=1075.603,172.288,-75.412,173.999,25.419,154.462
C08558=1075.609,172.536,-75.434,174.002,25.421,154.463
C08559=1075.614,172.785,-75.457,174.003,25.423,154.463
C08560=1075.620,173.034,-75.479,174.006,25.426,154.463
C08561=1075.626,173.284,-75.501,174.008,25.429,154.463
C08562=1075.631,173.532,-75.523,174.009,25.431,154.464
C08563=1075.636,173.781,-75.545,174.012,25.434,154.464
C08564=1075.643,174.030,-75.568,174.014,25.437,154.464
C08565=1075.648,174.279,-75.590,174.016,25.439,154.465
C08566=1075.654,174.528,-75.612,174.018,25.442,154.465
C08567=1075.660,174.777,-75.634,174.020,25.444,154.465
C08568=1075.666,175.058,-75.660,174.023,25.447,154.466
C08569=1075.672,175.339,-75.684,174.025,25.450,154.466
C08570=1075.679,175.620,-75.710,174.027,25.453,154.466
C08571=1075.685,175.900,-75.735,174.029,25.456,154.467
C08572=1075.691,176.150,-75.757,174.032,25.458,154.467
C08573=1075.696,176.399,-75.780,174.033,25.461,154.467
C08574=1075.702,176.648,-75.802,174.036,25.463,154.467
C08575=1075.708,176.897,-75.825,174.038,25.466,154.468
C08576=1075.713,177.146,-75.847,174.040,25.468,154.468
C08577=1075.719,177.395,-75.870,174.042,25.471,154.468
C08578=1075.725,177.643,-75.892,174.044,25.474,154.468
C08579=1075.731,177.893,-75.914,174.046,25.476,154.469
C08580=1075.736,178.142,-75.937,174.048,25.478,154.469
C08581=1075.741,178.391,-75.959,174.050,25.481,154.469
C08582=1075.748,178.639,-75.981,174.053,25.484,154.470
C08583=1075.753,178.888,-76.004,174.054,25.486,154.470
C08584=1075.759,179.138,-76.027,174.057,25.489,154.470
C08585=1075.765,179.386,-76.049,174.059,25.492,154.470
C08586=1075.771,179.635,-76.072,174.060,25.494,154.471
C08587=1075.776,179.884,-76.094,174.063,25.497,154.471
C08588=1075.782,180.133,-76.117,174.065,25.499,154.471
C08589=1075.787,180.382,-76.140,174.067,25.502,154.472
C08590=1075.793,180.631,-76.161,174.069,25.504,154.472
C08591=1075.799,180.880,-76.184,174.071,25.507,154.472
C08592=1075.805,181.129,-76.207,174.074,25.509,154.472
C08593=1075.811,181.378,-76.230,174.076,25.512,154.473
C08594=1075.817,181.627,-76.252,174.078,25.514,154.473
C08595=1075.823,181.876,-76.275,174.080,25.517,154.473
C08596=1075.828,182.125,-76.298,174.082,25.519,154.473
C08597=1075.833,182.373,-76.320,174.084,25.522,154.474
C08598=1075.840,182.621,-76.343,174.086,25.524,154.474
C08599=1075.845,182.871,-76.365,174.088,25.527,154.474
C08600=1075.851,183.120,-76.388,174.091,25.530,154.475
C08601=1075.857,183.369,-76.411,174.092,25.532,154.475
C08602=1075.862,183.617,-76.434,174.095,25.534,154.475
C08603=1075.869,183.866,-76.456,174.097,25.537,154.475
C08604=1075.875,184.115,-76.479,174.099,25.540,154.476
C08605=1075.880,184.365,-76.501,174.101,25.542,154.476
C08606=1075.886,184.613,-76.524,174.103,25.545,154.476
C08607=1075.892,184.862,-76.547,174.106,25.547,154.476
C08608=1075.897,185.111,-76.570,174.108,25.550,154.477
C08609=1075.903,185.360,-76.593,174.110,25.552,154.477
C08610=1075.909,185.609,-76.616,174.112,25.555,154.477
C08611=1075.914,185.857,-76.638,174.114,25.558,154.478
C08612=1075.919,186.106,-76.662,174.117,25.560,154.478
C08613=1075.925,186.355,-76.685,174.119,25.563,154.478
C08614=1075.930,186.604,-76.708,174.120,25.566,154.479
C08615=1075.936,186.853,-76.731,174.123,25.568,154.479
C08616=1075.941,187.102,-76.754,174.125,25.571,154.479
C08617=1075.947,187.351,-76.777,174.127,25.574,154.479
C08618=1075.953,187.600,-76.800,174.129,25.576,154.480
C08619=1075.958,187.848,-76.823,174.131,25.579,154.480
C08620=1075.963,188.097,-76.846,174.133,25.582,154.480
C08621=1075.968,188.346,-76.869,174.136,25.584,154.481
C08622=1075.974,188.595,-76.892,174.138,25.587,154.481
C08623=1075.980,188.844,-76.915,174.140,25.590,154.481
C08624=1075.986,189.093,-76.938,174.142,25.592,154.482
C08625=1075.991,189.342,-76.962,174.144,25.595,154.482
C08626=1075.997,189.591,-76.985,174.147,25.598,154.482
C08627=1076.002,189.839,-77.008,174.148,25.600,154.482
C08628=1076.008,190.088,-77.031,174.150,25.603,154.483
C08629=1076.013,190.338,-77.055,174.153,25.606,154.483
C08630=1076.019,190.586,-77.078,174.155,25.608,154.483
C08631=1076.025,190.835,-77.101,174.158,25.611,154.484
C08632=1076.031,191.116,-77.127,174.160,25.614,154.484
C08633=1076.037,191.397,-77.153,174.162,25.617,154.484
C08634=1076.043,191.677,-77.180,174.165,25.620,154.485
C08635=1076.049,191.958,-77.206,174.167,25.623,154.485
C08636=1076.055,192.206,-77.229,174.169,25.625,154.485
C08637=1076.060,192.455,-77.252,174.172,25.628,154.485
C08638=1076.066,192.704,-77.275,174.174,25.631,154.486
C08639=1076.071,192.953,-77.299,174.176,25.634,154.486
C08640=1076.077,193.202,-77.322,174.178,25.636,154.486
C08641=1076.083,193.450,-77.345,174.180,25.639,154.487
C08642=1076.089,193.700,-77.369,174.182,25.641,154.487
C08643=1076.095,193.949,-77.393,174.185,25.644,154.487
C08644=1076.100,194.198,-77.416,174.187,25.647,154.488
C08645=1076.105,194.447,-77.439,174.189,25.650,154.488
C08646=1076.111,194.695,-77.463,174.191,25.652,154.488
C08647=1076.117,194.944,-77.486,174.193,25.654,154.488
C08648=1076.122,195.193,-77.509,174.196,25.657,154.489
C08649=1076.128,195.441,-77.533,174.198,25.660,154.489
C08650=1076.134,195.690,-77.556,174.200,25.663,154.489
C08651=1076.139,195.940,-77.580,174.203,25.665,154.490
C08652=1076.145,196.188,-77.603,174.205,25.668,154.490
C08653=1076.151,196.437,-77.626,174.207,25.670,154.490
C08654=1076.156,196.685,-77.650,174.209,25.673,154.490
C08655=1076.162,196.935,-77.674,174.211,25.676,154.491
C08656=1076.168,197.184,-77.697,174.214,25.679,154.491
C08657=1076.173,197.432,-77.721,174.216,25.681,154.491
C08658=1076.179,197.681,-77.744,174.218,25.684,154.492
C08659=1076.184,197.930,-77.768,174.221,25.686,154.492
C08660=1076.190,198.179,-77.791,174.222,25.689,154.492
C08661=1076.196,198.427,-77.815,174.225,25.692,154.493
C08662=1076.202,198.677,-77.839,174.227,25.694,154.493
C08663=1076.208,198.925,-77.862,174.229,25.697,154.493
C08664=1076.213,199.174,-77.886,174.232,25.700,154.493
C08665=1076.219,199.423,-77.910,174.234,25.702,154.494
C08666=1076.225,199.671,-77.933,174.237,25.705,154.494
C08667=1076.230,199.921,-77.957,174.239,25.707,154.494
C08668=1076.236,200.169,-77.981,174.240,25.710,154.495
C08669=1076.241,200.418,-78.004,174.243,25.713,154.495
C08670=1076.247,200.667,-78.028,174.245,25.715,154.495
C08671=1076.253,200.916,-78.051,174.247,25.718,154.495
C08672=1076.259,201.165,-78.076,174.250,25.721,154.496
C08673=1076.265,201.413,-78.099,174.252,25.723,154.496
C08674=1076.270,201.662,-78.123,174.254,25.726,154.496
C08675=1076.276,201.911,-78.146,174.257,25.729,154.497
C08676=1076.282,202.160,-78.171,174.259,25.731,154.497
C08677=1076.288,202.409,-78.194,174.262,25.734,154.497
C08678=1076.293,202.657,-78.218,174.263,25.736,154.497
C08679=1076.299,202.906,-78.242,174.265,25.739,154.498
C08680=1076.304,203.155,-78.265,174.268,25.742,154.498
C08681=1076.310,203.404,-78.290,174.270,25.745,154.498
C08682=1076.316,203.652,-78.314,174.273,25.747,154.499
C08683=1076.321,203.901,-78.338,174.275,25.750,154.499
C08684=1076.326,204.150,-78.362,174.277,25.753,154.499
C08685=1076.333,204.399,-78.386,174.280,25.755,154.500
C08686=1076.338,204.648,-78.410,174.282,25.759,154.500
C08687=1076.344,204.896,-78.434,174.284,25.761,154.500
C08688=1076.350,205.145,-78.458,174.287,25.764,154.500
C08689=1076.355,205.394,-78.481,174.289,25.767,154.501
C08690=1076.360,205.643,-78.506,174.291,25.769,154.501
C08691=1076.366,205.891,-78.530,174.293,25.772,154.501
C08692=1076.372,206.140,-78.554,174.295,25.774,154.502
C08693=1076.377,206.389,-78.578,174.298,25.777,154.502
C08694=1076.383,206.638,-78.603,174.300,25.780,154.502
C08695=1076.389,206.886,-78.626,174.302,25.783,154.503
C08696=1076.413,207.924,-78.727,174.417,25.843,154.502
C08697=1076.422,208.332,-78.768,174.420,25.849,154.503
C08698=1076.431,208.741,-78.808,174.424,25.855,154.504
C08699=1076.440,209.149,-78.849,174.427,25.862,154.505
C08700=1076.450,209.557,-78.890,174.431,25.867,154.506
C08701=1076.456,209.806,-78.914,174.433,25.871,154.506
C08702=1076.462,210.055,-78.940,174.435,25.875,154.507
C08703=1076.467,210.304,-78.964,174.438,25.878,154.507
C08704=1076.473,210.552,-78.989,174.440,25.882,154.508
C08705=1076.479,210.801,-79.013,174.442,25.886,154.508
C08706=1076.485,211.050,-79.039,174.444,25.889,154.509
C08707=1076.490,211.298,-79.063,174.446,25.893,154.509
C08708=1076.496,211.547,-79.088,174.448,25.897,154.510
C08709=1076.502,211.796,-79.113,174.450,25.900,154.510
C08710=1076.507,212.044,-79.138,174.453,25.904,154.511
C08711=1076.513,212.294,-79.163,174.455,25.907,154.511
C08712=1076.519,212.542,-79.188,174.457,25.911,154.512
C08713=1076.525,212.790,-79.213,174.459,25.915,154.513
C08714=1076.531,213.040,-79.238,174.461,25.918,154.513
C08715=1076.536,213.288,-79.263,174.463,25.922,154.514
C08716=1076.542,213.537,-79.288,174.465,25.926,154.514
C08717=1076.547,213.785,-79.313,174.468,25.930,154.515
C08718=1076.553,214.034,-79.339,174.470,25.933,154.515
C08719=1076.559,214.283,-79.363,174.472,25.937,154.516
C08720=1076.564,214.531,-79.389,174.474,25.941,154.516
C08721=1076.570,214.780,-79.414,174.476,25.944,154.517
C08722=1076.576,215.029,-79.439,174.478,25.948,154.517
C08723=1076.582,215.277,-79.464,174.481,25.952,154.518
C08724=1076.587,215.526,-79.490,174.483,25.955,154.518
C08725=1076.594,215.775,-79.515,174.485,25.959,154.519
C08726=1076.599,216.024,-79.539,174.488,25.963,154.519
C08727=1076.605,216.272,-79.565,174.490,25.966,154.520
C08728=1076.610,216.521,-79.590,174.492,25.970,154.520
C08729=1076.616,216.769,-79.615,174.495,25.974,154.521
C08730=1076.622,217.018,-79.641,174.497,25.977,154.521
C08731=1076.627,217.267,-79.666,174.499,25.981,154.522
C08732=1076.633,217.515,-79.691,174.501,25.985,154.523
C08733=1076.639,217.764,-79.716,174.503,25.989,154.523
C08734=1076.645,218.013,-79.742,174.505,25.992,154.524
C08735=1076.650,218.261,-79.767,174.507,25.996,154.524
C08736=1076.657,218.510,-79.793,174.510,26.000,154.525
C08737=1076.662,218.759,-79.818,174.512,26.003,154.525
C08738=1076.668,219.008,-79.843,174.514,26.007,154.526
C08739=1076.674,219.256,-79.868,174.516,26.010,154.526
C08740=1076.679,219.505,-79.894,174.518,26.014,154.527
C08741=1076.685,219.754,-79.919,174.521,26.018,154.527
C08742=1076.691,220.002,-79.945,174.524,26.021,154.528
C08743=1076.697,220.251,-79.971,174.526,26.025,154.528
C08744=1076.702,220.499,-79.996,174.528,26.028,154.529
C08745=1076.709,220.748,-80.021,174.530,26.032,154.529
C08746=1076.714,220.997,-80.047,174.532,26.036,154.530
C08747=1076.720,221.246,-80.072,174.535,26.039,154.530
C08748=1076.726,221.495,-80.098,174.537,26.043,154.531
C08749=1076.736,221.907,-80.140,174.540,26.049,154.532
C08750=1076.744,222.319,-80.183,174.544,26.055,154.533
C08751=1076.754,222.732,-80.225,174.549,26.061,154.533
C08752=1076.764,223.144,-80.268,174.552,26.068,154.534
C08753=1076.770,223.393,-80.293,174.554,26.071,154.535
C08754=1076.775,223.642,-80.319,174.556,26.075,154.535
C08755=1076.781,223.891,-80.345,174.559,26.079,154.536
C08756=1076.786,224.139,-80.370,174.561,26.082,154.536
C08757=1076.792,224.387,-80.397,174.563,26.086,154.537
C08758=1076.798,224.636,-80.422,174.565,26.089,154.537
C08759=1076.804,224.885,-80.448,174.567,26.093,154.538
C08760=1076.809,225.134,-80.474,174.570,26.097,154.538
C08761=1076.815,225.382,-80.499,174.573,26.101,154.539
C08762=1076.821,225.631,-80.526,174.575,26.104,154.540
C08763=1076.827,225.879,-80.551,174.577,26.108,154.540
C08764=1076.832,226.128,-80.577,174.579,26.111,154.541
C08765=1076.838,226.377,-80.603,174.581,26.115,154.541
C08766=1076.844,226.625,-80.629,174.584,26.119,154.542
C08767=1076.850,226.874,-80.655,174.586,26.122,154.542
C08768=1076.855,227.123,-80.681,174.588,26.126,154.543
C08769=1076.862,227.371,-80.707,174.591,26.130,154.543
C08770=1076.867,227.620,-80.733,174.593,26.133,154.544
C08771=1076.873,227.869,-80.759,174.595,26.137,154.544
C08772=1076.879,228.116,-80.784,174.598,26.141,154.545
C08773=1076.884,228.365,-80.810,174.600,26.144,154.545
C08774=1076.889,228.614,-80.836,174.602,26.148,154.546
C08775=1076.896,228.862,-80.862,174.604,26.151,154.546
C08776=1076.901,229.111,-80.888,174.607,26.155,154.547
C08777=1076.907,229.359,-80.915,174.610,26.159,154.547
C08778=1076.913,229.608,-80.940,174.612,26.163,154.548
C08779=1076.919,229.856,-80.967,174.614,26.166,154.548
C08780=1076.925,230.105,-80.993,174.616,26.170,154.549
C08781=1076.931,230.354,-81.018,174.618,26.173,154.549
C08782=1076.937,230.602,-81.045,174.620,26.177,154.550
C08783=1076.942,230.851,-81.071,174.624,26.181,154.550
C08784=1076.948,231.100,-81.097,174.626,26.185,154.551
C08785=1076.953,231.349,-81.123,174.628,26.188,154.551
C08786=1076.959,231.597,-81.150,174.630,26.192,154.552
C08787=1076.966,231.845,-81.176,174.632,26.195,154.553
C08788=1076.971,232.094,-81.202,174.635,26.199,154.553
C08789=1076.977,232.343,-81.229,174.637,26.203,154.554
C08790=1076.982,232.592,-81.254,174.640,26.206,154.554
C08791=1076.988,232.840,-81.281,174.642,26.210,154.555
C08792=1076.994,233.088,-81.308,174.644,26.214,154.555
C08793=1076.999,233.337,-81.334,174.646,26.217,154.556
C08794=1077.005,233.586,-81.360,174.649,26.221,154.556
C08795=1077.011,233.835,-81.386,174.651,26.224,154.557
C08796=1077.016,234.083,-81.413,174.654,26.228,154.557
C08797=1077.022,234.331,-81.440,174.656,26.232,154.558
C08798=1077.028,234.580,-81.466,174.658,26.236,154.558
C08799=1077.033,234.829,-81.492,174.661,26.239,154.559
C08800=1077.039,235.077,-81.519,174.663,26.243,154.559
C08801=1077.049,235.481,-81.562,174.667,26.249,154.560
C08802=1077.058,235.885,-81.604,174.671,26.255,154.561
C08803=1077.067,236.289,-81.648,174.675,26.261,154.562
C08804=1077.077,236.694,-81.691,174.678,26.267,154.563
C08805=1077.082,236.942,-81.717,174.681,26.270,154.563
C08806=1077.088,237.190,-81.744,174.683,26.274,154.564
C08807=1077.094,237.439,-81.771,174.686,26.278,154.564
C08808=1077.100,237.688,-81.798,174.688,26.282,154.565
C08809=1077.106,237.937,-81.824,174.690,26.285,154.565
C08810=1077.111,238.185,-81.850,174.693,26.289,154.566
C08811=1077.117,238.433,-81.877,174.695,26.292,154.566
C08812=1077.123,238.682,-81.903,174.698,26.296,154.567
C08813=1077.129,238.930,-81.930,174.700,26.300,154.567
C08814=1077.134,239.179,-81.957,174.702,26.303,154.568
C08815=1077.140,239.428,-81.984,174.705,26.307,154.568
C08816=1077.146,239.676,-82.011,174.707,26.311,154.569
C08817=1077.152,239.925,-82.038,174.710,26.315,154.569
C08818=1077.158,240.173,-82.064,174.712,26.318,154.570
C08819=1077.163,240.421,-82.091,174.714,26.322,154.570
C08820=1077.169,240.670,-82.118,174.717,26.325,154.571
C08821=1077.175,240.919,-82.145,174.720,26.329,154.571
C08822=1077.181,241.167,-82.171,174.722,26.333,154.572
C08823=1077.186,241.416,-82.199,174.724,26.336,154.573
C08824=1077.192,241.664,-82.225,174.726,26.340,154.573
C08825=1077.198,241.912,-82.252,174.729,26.344,154.574
C08826=1077.204,242.162,-82.279,174.732,26.347,154.574
C08827=1077.210,242.410,-82.305,174.734,26.351,154.575
C08828=1077.216,242.658,-82.332,174.736,26.355,154.575
C08829=1077.221,242.907,-82.359,174.738,26.358,154.576
C08830=1077.227,243.155,-82.387,174.741,26.362,154.576
C08831=1077.233,243.404,-82.414,174.744,26.366,154.577
C08832=1077.238,243.652,-82.441,174.746,26.369,154.577
C08833=1077.244,243.901,-82.468,174.748,26.373,154.578
C08834=1077.250,244.149,-82.494,174.751,26.377,154.578
C08835=1077.255,244.397,-82.522,174.753,26.381,154.579
C08836=1077.262,244.646,-82.549,174.756,26.384,154.579
C08837=1077.267,244.895,-82.576,174.758,26.388,154.580
C08838=1077.272,245.143,-82.603,174.761,26.392,154.580
C08839=1077.278,245.391,-82.630,174.763,26.395,154.581
C08840=1077.284,245.639,-82.657,174.765,26.399,154.581
C08841=1077.290,245.889,-82.685,174.768,26.403,154.582
C08842=1077.296,246.137,-82.711,174.771,26.407,154.583
C08843=1077.301,246.385,-82.739,174.773,26.410,154.583
C08844=1077.307,246.634,-82.766,174.775,26.414,154.584
C08845=1077.313,246.883,-82.793,174.777,26.417,154.584
C08846=1077.318,247.131,-82.821,174.781,26.421,154.585
C08847=1077.324,247.379,-82.848,174.783,26.425,154.585
C08848=1077.330,247.628,-82.875,174.785,26.428,154.586
C08849=1077.336,247.876,-82.903,174.787,26.432,154.586
C08850=1077.341,248.125,-82.930,174.790,26.436,154.587
C08851=1077.346,248.373,-82.958,174.792,26.440,154.587
C08852=1077.353,248.622,-82.985,174.795,26.443,154.588
C08853=1077.361,249.019,-83.029,174.798,26.449,154.589
C08854=1077.370,249.416,-83.073,174.803,26.456,154.590
C08855=1077.379,249.814,-83.116,174.807,26.462,154.590
C08856=1077.388,250.211,-83.160,174.811,26.467,154.591
C08857=1077.394,250.460,-83.189,174.813,26.471,154.592
C08858=1077.400,250.709,-83.215,174.816,26.475,154.592
C08859=1077.405,250.957,-83.243,174.818,26.478,154.593
C08860=1077.412,251.205,-83.271,174.820,26.482,154.593
C08861=1077.417,251.454,-83.298,174.823,26.486,154.594
C08862=1077.422,251.702,-83.326,174.826,26.490,154.595
C08863=1077.429,251.951,-83.353,174.828,26.494,154.595
C08864=1077.434,252.199,-83.381,174.830,26.497,154.596
C08865=1077.440,252.448,-83.409,174.833,26.501,154.596
C08866=1077.446,252.696,-83.436,174.835,26.505,154.597
C08867=1077.451,252.944,-83.464,174.838,26.508,154.597
C08868=1077.457,253.193,-83.492,174.841,26.512,154.598
C08869=1077.463,253.441,-83.519,174.843,26.516,154.598
C08870=1077.468,253.689,-83.547,174.845,26.519,154.599
C08871=1077.474,253.938,-83.575,174.847,26.523,154.599
C08872=1077.480,254.186,-83.603,174.851,26.527,154.600
C08873=1077.486,254.435,-83.630,174.853,26.531,154.600
C08874=1077.491,254.683,-83.658,174.855,26.534,154.601
C08875=1077.498,254.932,-83.686,174.858,26.538,154.601
C08876=1077.503,255.180,-83.714,174.861,26.542,154.602
C08877=1077.508,255.428,-83.741,174.863,26.545,154.602
C08878=1077.515,255.677,-83.769,174.866,26.549,154.603
C08879=1077.520,255.925,-83.797,174.868,26.553,154.603
C08880=1077.526,256.174,-83.825,174.870,26.556,154.604
C08881=1077.532,256.421,-83.853,174.874,26.560,154.605
C08882=1077.538,256.670,-83.881,174.876,26.564,154.605
C08883=1077.544,256.918,-83.909,174.878,26.567,154.606
C08884=1077.549,257.167,-83.936,174.881,26.572,154.606
C08885=1077.555,257.415,-83.964,174.883,26.575,154.607
C08886=1077.561,257.664,-83.992,174.886,26.579,154.607
C08887=1077.567,257.912,-84.020,174.889,26.583,154.608
C08888=1077.572,258.161,-84.048,174.891,26.586,154.608
C08889=1077.579,258.409,-84.076,174.893,26.590,154.609
C08890=1077.585,258.657,-84.104,174.896,26.594,154.609
C08891=1077.590,258.906,-84.132,174.899,26.597,154.610
C08892=1077.596,259.154,-84.160,174.901,26.601,154.610
C08893=1077.602,259.402,-84.188,174.904,26.605,154.611
C08894=1077.608,259.651,-84.216,174.906,26.608,154.611
C08895=1077.614,259.899,-84.244,174.909,26.612,154.612
C08896=1077.619,260.147,-84.272,174.912,26.616,154.612
C08897=1077.626,260.396,-84.300,174.914,26.619,154.613
C08898=1077.632,260.644,-84.329,174.917,26.623,154.613
C08899=1077.637,260.892,-84.357,174.919,26.627,154.614
C08900=1077.643,261.141,-84.385,174.922,26.630,154.615
C08901=1077.649,261.389,-84.414,174.925,26.634,154.615
C08902=1077.655,261.637,-84.441,174.927,26.637,154.616
C08903=1077.661,261.886,-84.469,174.929,26.641,154.616
C08904=1077.667,262.134,-84.497,174.933,26.645,154.617
C08905=1077.677,262.529,-84.543,174.936,26.651,154.617
C08906=1077.686,262.924,-84.588,174.940,26.656,154.618
C08907=1077.695,263.319,-84.632,174.945,26.662,154.619
C08908=1077.704,263.714,-84.677,174.949,26.668,154.620
C08909=1077.711,263.962,-84.706,174.952,26.672,154.620
C08910=1077.717,264.211,-84.735,174.954,26.676,154.621
C08911=1077.722,264.459,-84.763,174.956,26.679,154.622
C08912=1077.728,264.707,-84.792,174.959,26.683,154.622
C08913=1077.733,264.955,-84.820,174.962,26.687,154.623
C08914=1077.739,265.204,-84.848,174.965,26.691,154.623
C08915=1077.746,265.452,-84.877,174.967,26.694,154.624
C08916=1077.751,265.700,-84.905,174.969,26.698,154.624
C08917=1077.757,265.948,-84.934,174.973,26.702,154.625
C08918=1077.762,266.197,-84.963,174.975,26.706,154.625
C08919=1077.768,266.445,-84.991,174.977,26.709,154.626
C08920=1077.774,266.693,-85.020,174.980,26.713,154.626
C08921=1077.780,266.942,-85.048,174.982,26.717,154.627
C08922=1077.786,267.189,-85.077,174.986,26.721,154.627
C08923=1077.792,267.438,-85.105,174.988,26.725,154.628
C08924=1077.798,267.686,-85.134,174.990,26.728,154.629
C08925=1077.803,267.934,-85.162,174.993,26.732,154.629
C08926=1077.809,268.183,-85.192,174.995,26.736,154.630
C08927=1077.815,268.432,-85.220,174.999,26.740,154.630
C08928=1077.821,268.680,-85.249,175.001,26.743,154.631
C08929=1077.826,268.928,-85.277,175.004,26.747,154.631
C08930=1077.832,269.176,-85.306,175.006,26.751,154.632
C08931=1077.838,269.424,-85.336,175.008,26.754,154.632
C08932=1077.844,269.673,-85.364,175.012,26.758,154.633
C08933=1077.850,269.921,-85.393,175.014,26.762,154.633
C08934=1077.855,270.169,-85.421,175.017,26.766,154.634
C08935=1077.861,270.418,-85.451,175.019,26.770,154.635
C08936=1077.867,270.666,-85.480,175.022,26.773,154.635
C08937=1077.873,270.914,-85.508,175.025,26.777,154.636
C08938=1077.879,271.162,-85.537,175.027,26.781,154.636
C08939=1077.884,271.410,-85.566,175.030,26.785,154.637
C08940=1077.891,271.659,-85.596,175.032,26.789,154.637
C08941=1077.897,271.907,-85.624,175.036,26.792,154.638
C08942=1077.901,272.155,-85.653,175.038,26.796,154.638
C08943=1077.908,272.403,-85.682,175.041,26.800,154.639
C08944=1077.914,272.651,-85.711,175.043,26.804,154.640
C08945=1077.919,272.900,-85.740,175.045,26.807,154.640
C08946=1077.925,273.149,-85.769,175.049,26.811,154.641
C08947=1077.931,273.396,-85.798,175.051,26.815,154.641
C08948=1077.937,273.644,-85.827,175.054,26.819,154.642
C08949=1077.943,273.893,-85.857,175.056,26.823,154.642
C08950=1077.948,274.141,-85.886,175.060,26.826,154.643
C08951=1077.954,274.390,-85.914,175.062,26.830,154.643
C08952=1077.960,274.638,-85.944,175.065,26.834,154.644
C08953=1077.965,274.886,-85.973,175.067,26.838,154.644
C08954=1077.972,275.134,-86.002,175.070,26.842,154.645
C08955=1077.977,275.382,-86.031,175.073,26.846,154.646
C08956=1077.983,275.630,-86.061,175.075,26.849,154.646
C08957=1077.993,276.028,-86.108,175.080,26.855,154.647
C08958=1078.001,276.427,-86.154,175.084,26.862,154.648
C08959=1078.011,276.825,-86.202,175.088,26.867,154.649
C08960=1078.020,277.222,-86.248,175.093,26.874,154.650
C08961=1078.026,277.471,-86.278,175.095,26.878,154.650
C08962=1078.032,277.719,-86.307,175.098,26.882,154.651
C08963=1078.038,277.967,-86.337,175.100,26.885,154.651
C08964=1078.043,278.216,-86.366,175.104,26.889,154.652
C08965=1078.050,278.463,-86.396,175.106,26.893,154.653
C08966=1078.055,278.711,-86.426,175.109,26.897,154.653
C08967=1078.062,278.960,-86.455,175.111,26.901,154.654
C08968=1078.067,279.208,-86.484,175.114,26.905,154.654
C08969=1078.073,279.456,-86.513,175.117,26.908,154.655
C08970=1078.078,279.704,-86.543,175.120,26.912,154.655
C08971=1078.084,279.952,-86.573,175.122,26.916,154.656
C08972=1078.090,280.200,-86.602,175.125,26.920,154.656
C08973=1078.096,280.448,-86.632,175.128,26.924,154.657
C08974=1078.102,280.696,-86.661,175.131,26.928,154.658
C08975=1078.108,280.945,-86.690,175.133,26.932,154.658
C08976=1078.113,281.193,-86.721,175.136,26.935,154.659
C08977=1078.119,281.441,-86.750,175.138,26.939,154.659
C08978=1078.125,281.689,-86.779,175.142,26.943,154.660
C08979=1078.131,281.937,-86.810,175.144,26.947,154.661
C08980=1078.136,282.186,-86.839,175.147,26.951,154.661
C08981=1078.142,282.434,-86.869,175.149,26.955,154.662
C08982=1078.148,282.682,-86.899,175.152,26.959,154.662
C08983=1078.154,282.930,-86.928,175.155,26.962,154.663
C08984=1078.160,283.178,-86.959,175.158,26.967,154.663
C08985=1078.165,283.426,-86.988,175.160,26.970,154.664
C08986=1078.171,283.675,-87.018,175.163,26.975,154.665
C08987=1078.177,283.922,-87.048,175.165,26.978,154.665
C08988=1078.183,284.171,-87.077,175.169,26.982,154.666
C08989=1078.189,284.418,-87.108,175.171,26.986,154.666
C08990=1078.194,284.667,-87.137,175.174,26.990,154.667
C08991=1078.200,284.915,-87.168,175.176,26.994,154.667
C08992=1078.206,285.163,-87.197,175.180,26.998,154.668
C08993=1078.211,285.411,-87.228,175.182,27.002,154.669
C08994=1078.218,285.660,-87.257,175.185,27.005,154.669
C08995=1078.224,285.908,-87.288,175.188,27.010,154.670
C08996=1078.230,286.155,-87.318,175.190,27.013,154.670
C08997=1078.235,286.404,-87.348,175.193,27.018,154.671
C08998=1078.241,286.652,-87.378,175.196,27.021,154.671
C08999=1078.247,286.900,-87.408,175.199,27.025,154.672
C09000=1078.253,287.148,-87.438,175.201,27.029,154.673
C09001=1078.259,287.395,-87.468,175.204,27.033,154.673
C09002=1078.265,287.644,-87.497,175.207,27.037,154.674
C09003=1078.271,287.892,-87.528,175.210,27.041,154.674
C09004=1078.277,288.140,-87.558,175.213,27.045,154.675
C09005=1078.282,288.389,-87.588,175.215,27.048,154.675
C09006=1078.288,288.637,-87.618,175.218,27.053,154.676
C09007=1078.294,288.884,-87.649,175.221,27.056,154.677
C09008=1078.300,289.132,-87.679,175.224,27.061,154.677
C09009=1078.310,289.541,-87.728,175.229,27.067,154.678
C09010=1078.320,289.948,-87.778,175.233,27.073,154.679
C09011=1078.329,290.356,-87.829,175.237,27.080,154.680
C09012=1078.339,290.764,-87.878,175.242,27.086,154.681
C09013=1078.344,291.012,-87.908,175.245,27.090,154.682
C09014=1078.350,291.260,-87.939,175.248,27.094,154.682
C09015=1078.356,291.508,-87.969,175.250,27.098,154.683
C09016=1078.362,291.756,-87.999,175.254,27.102,154.683
C09017=1078.368,292.004,-88.030,175.256,27.106,154.684
C09018=1078.373,292.252,-88.061,175.259,27.110,154.685
C09019=1078.379,292.500,-88.091,175.261,27.114,154.685
C09020=1078.385,292.748,-88.122,175.264,27.118,154.686
C09021=1078.391,292.996,-88.152,175.268,27.122,154.686
C09022=1078.397,293.244,-88.183,175.270,27.126,154.687
C09023=1078.403,293.492,-88.213,175.273,27.130,154.688
C09024=1078.408,293.740,-88.244,175.276,27.134,154.688
C09025=1078.414,293.988,-88.274,175.278,27.138,154.689
C09026=1078.420,294.237,-88.305,175.282,27.142,154.690
C09027=1078.426,294.485,-88.335,175.284,27.146,154.690
C09028=1078.432,294.732,-88.366,175.287,27.150,154.691
C09029=1078.438,294.980,-88.396,175.290,27.154,154.691
C09030=1078.444,295.229,-88.427,175.292,27.158,154.692
C09031=1078.449,295.477,-88.458,175.296,27.162,154.692
C09032=1078.456,295.724,-88.489,175.298,27.166,154.693
C09033=1078.462,295.973,-88.520,175.301,27.170,154.694
C09034=1078.467,296.221,-88.551,175.304,27.174,154.694
C09035=1078.473,296.468,-88.581,175.306,27.178,154.695
C09036=1078.479,296.717,-88.612,175.310,27.182,154.695
C09037=1078.485,296.964,-88.643,175.313,27.186,154.696
C09038=1078.490,297.212,-88.674,175.315,27.190,154.697
C09039=1078.497,297.461,-88.704,175.318,27.194,154.697
C09040=1078.503,297.709,-88.735,175.321,27.199,154.698
C09041=1078.508,297.956,-88.766,175.324,27.203,154.699
C09042=1078.514,298.204,-88.797,175.327,27.207,154.699
C09043=1078.520,298.453,-88.828,175.330,27.211,154.700
C09044=1078.526,298.700,-88.859,175.332,27.215,154.700
C09045=1078.531,298.948,-88.890,175.335,27.219,154.701
C09046=1078.537,299.196,-88.922,175.338,27.223,154.702
C09047=1078.543,299.444,-88.952,175.341,27.227,154.702
C09048=1078.548,299.692,-88.983,175.344,27.231,154.703
C09049=1078.554,299.940,-89.014,175.346,27.235,154.704
C09050=1078.559,300.188,-89.046,175.349,27.240,154.704
C09051=1078.566,300.436,-89.077,175.352,27.244,154.705
C09052=1078.571,300.684,-89.108,175.355,27.248,154.706
C09053=1078.577,300.932,-89.139,175.358,27.252,154.706
C09054=1078.582,301.180,-89.170,175.361,27.257,154.707
C09055=1078.588,301.428,-89.202,175.363,27.260,154.707
C09056=1078.594,301.676,-89.233,175.367,27.264,154.708
C09057=1078.600,301.923,-89.264,175.370,27.269,154.709
C09058=1078.606,302.172,-89.295,175.372,27.273,154.709
C09059=1078.611,302.419,-89.327,175.375,27.277,154.710
C09060=1078.617,302.668,-89.359,175.378,27.281,154.711
C09061=1078.623,302.878,-89.385,175.381,27.285,154.711
C09062=1078.627,303.089,-89.411,175.383,27.288,154.712
C09063=1078.632,303.300,-89.438,175.385,27.292,154.712
C09064=1078.637,303.512,-89.465,175.388,27.295,154.713
C09065=1078.642,303.723,-89.491,175.391,27.299,154.713
C09066=1078.647,303.935,-89.518,175.393,27.302,154.714
C09067=1078.652,304.145,-89.545,175.395,27.306,154.715
C09068=1078.657,304.356,-89.572,175.398,27.310,154.715
C09069=1078.663,304.604,-89.603,175.401,27.314,154.716
C09070=1078.669,304.853,-89.634,175.403,27.318,154.716
C09071=1078.674,305.100,-89.666,175.406,27.322,154.717
C09072=1078.681,305.348,-89.697,175.410,27.326,154.718
C09073=1078.686,305.595,-89.729,175.413,27.330,154.718
C09074=1078.692,305.844,-89.760,175.415,27.334,154.719
C09075=1078.698,306.091,-89.791,175.418,27.339,154.719
C09076=1078.704,306.340,-89.823,175.421,27.343,154.720
C09077=1078.709,306.587,-89.855,175.424,27.347,154.721
C09078=1078.716,306.835,-89.887,175.427,27.351,154.721
C09079=1078.722,307.083,-89.918,175.430,27.355,154.722
C09080=1078.727,307.331,-89.950,175.433,27.360,154.723
C09081=1078.733,307.579,-89.981,175.435,27.364,154.723
C09082=1078.739,307.827,-90.013,175.438,27.368,154.724
C09083=1078.745,308.075,-90.045,175.442,27.372,154.725
C09084=1078.751,308.323,-90.076,175.445,27.376,154.725
C09085=1078.757,308.571,-90.108,175.447,27.380,154.726
C09086=1078.763,308.818,-90.139,175.450,27.385,154.727
